QRS_NEXT_CUT()
PTP {E1 28976.919,E2 28976.919}
PTP {X 0,Y 607.89,A -85,B 0,C 180,E1 28976.919,E2 28976.919,E3 0,E4 0,E5 0,E6 0}
QRS_SPEED_INIT()
LIN {X 0,Y 607.89,Z 1319.5,A -85,B 0,C 180,E1 28976.919,E2 28976.919,E3 0,E4 0,E5 0,E6 0} C_VEL
LIN {X 0,Y 607.89,Z 669.091,A -85,B 0,C 180,E1 28976.919,E2 28976.919} C_VEL
LIN {X 0,Y 607.89,Z 661.015,A -85,B 0,C 180,E1 28976.919,E2 28976.919} C_VEL
LIN {X 0,Y 607.896,Z 659.015,A -85,B 0,C 180,E1 28976.73,E2 28976.73} C_VEL
LIN {X 0,Y 607.914,Z 659.013,A -85,B 0,C 180,E1 28973.578,E2 28973.578} C_VEL
LIN {X 0,Y 607.913,Z 659.015,A -85,B 0,C 180,E1 28970.342,E2 28970.342} C_VEL
LIN {X 0,Y 607.906,Z 659.015,A -85,B 0,C 180,E1 28967.171,E2 28967.171} C_VEL
LIN {X 0,Y 607.906,Z 659.013,A -85,B 0,C 180,E1 28963.959,E2 28963.959} C_VEL
LIN {X 0,Y 607.896,Z 659.013,A -85,B 0,C 180,E1 28960.751,E2 28960.751} C_VEL
LIN {X 0,Y 607.9,Z 659.012,A -85,B 0,C 180,E1 28957.67,E2 28957.67} C_VEL
LIN {X 0,Y 607.904,Z 659.011,A -85,B 0,C 180,E1 28954.473,E2 28954.473} C_VEL
LIN {X 0,Y 607.904,Z 659.009,A -85,B 0,C 180,E1 28951.241,E2 28951.241} C_VEL
LIN {X 0,Y 607.906,Z 659.01,A -85,B 0,C 180,E1 28948.021,E2 28948.021} C_VEL
LIN {X 0,Y 607.908,Z 659.009,A -85,B 0,C 180,E1 28944.828,E2 28944.828} C_VEL
LIN {X 0,Y 607.911,Z 659.01,A -85,B 0,C 180,E1 28941.526,E2 28941.526} C_VEL
LIN {X 0,Y 607.907,Z 659.011,A -85,B 0,C 180,E1 28938.306,E2 28938.306} C_VEL
LIN {X 0,Y 607.917,Z 659.013,A -85,B 0,C 180,E1 28935.009,E2 28935.009} C_VEL
LIN {X 0,Y 607.911,Z 659.016,A -85,B 0,C 180,E1 28931.768,E2 28931.768} C_VEL
LIN {X 0,Y 607.904,Z 659.015,A -85,B 0,C 180,E1 28928.562,E2 28928.562} C_VEL
LIN {X 0,Y 607.904,Z 659.014,A -85,B 0,C 180,E1 28925.376,E2 28925.376} C_VEL
LIN {X 0,Y 607.916,Z 659.13,A -85,B 0,C 180,E1 28924.285,E2 28924.285} C_VEL
LIN {X 0,Y 607.915,Z 707.559,A -85,B 0,C 180,E1 28921.204,E2 28921.204} C_VEL
LIN {X 0,Y 607.914,Z 757.754,A -85,B 0,C 180,E1 28918.113,E2 28918.113} C_VEL
LIN {X 0,Y 607.895,Z 765.812,A -85,B 0,C 180,E1 28917.641,E2 28917.641} C_VEL
LIN {X 0,Y 607.908,Z 1003.67,A -85,B 0,C 180,E1 28914.573,E2 28914.573} C_VEL
LIN {X 0,Y 607.919,Z 1031.222,A -85,B 0,C 180,E1 28914.175,E2 28914.175} C_VEL
LIN {X 0,Y 607.917,Z 1051.471,A -85,B 0,C 180,E1 28913.711,E2 28913.711} C_VEL
LIN {X 0,Y 607.906,Z 1071.416,A -85,B 0,C 180,E1 28913.07,E2 28913.07} C_VEL
LIN {X 0,Y 607.906,Z 1090.488,A -85,B 0,C 180,E1 28912.278,E2 28912.278} C_VEL
LIN {X 0,Y 607.918,Z 1109.332,A -85,B 0,C 180,E1 28911.314,E2 28911.314} C_VEL
LIN {X 0,Y 607.917,Z 1127.307,A -85,B 0,C 180,E1 28910.205,E2 28910.205} C_VEL
LIN {X 0,Y 607.912,Z 1144.273,A -85,B 0,C 180,E1 28908.963,E2 28908.963} C_VEL
LIN {X 0,Y 607.917,Z 1160.452,A -85,B 0,C 180,E1 28907.566,E2 28907.566} C_VEL
LIN {X 0,Y 607.913,Z 1175.45,A -85,B 0,C 180,E1 28906.04,E2 28906.04} C_VEL
LIN {X 0,Y 607.913,Z 1189.435,A -85,B 0,C 180,E1 28904.36,E2 28904.36} C_VEL
LIN {X 0,Y 607.909,Z 1201.499,A -85,B 0,C 180,E1 28902.635,E2 28902.635} C_VEL
LIN {X 0,Y 607.917,Z 1211.62,A -85,B 0,C 180,E1 28900.902,E2 28900.902} C_VEL
LIN {X 0,Y 607.904,Z 1220.371,A -85,B 0,C 180,E1 28899.084,E2 28899.084} C_VEL
LIN {X 0,Y 607.901,Z 1227.349,A -85,B 0,C 180,E1 28897.275,E2 28897.275} C_VEL
LIN {X 0,Y 607.911,Z 1232.888,A -85,B 0,C 180,E1 28895.379,E2 28895.379} C_VEL
LIN {X 0,Y 607.905,Z 1236.665,A -85,B 0,C 180,E1 28893.489,E2 28893.489} C_VEL
LIN {X 0,Y 607.904,Z 1238.841,A -85,B 0,C 180,E1 28891.602,E2 28891.602} C_VEL
LIN {X 0,Y 607.904,Z 1239.45,A -85,B 0,C 180,E1 28889.717,E2 28889.717} C_VEL
LIN {X 0,Y 607.919,Z 1238.497,A -85,B 0,C 180,E1 28887.832,E2 28887.832} C_VEL
LIN {X 0,Y 607.916,Z 1235.709,A -85,B 0,C 180,E1 28885.85,E2 28885.85} C_VEL
LIN {X 0,Y 607.91,Z 1231.354,A -85,B 0,C 180,E1 28883.957,E2 28883.957} C_VEL
LIN {X 0,Y 607.904,Z 1225.285,A -85,B 0,C 180,E1 28882.058,E2 28882.058} C_VEL
LIN {X 0,Y 607.911,Z 1217.814,A -85,B 0,C 180,E1 28880.246,E2 28880.246} C_VEL
LIN {X 0,Y 607.907,Z 1208.471,A -85,B 0,C 180,E1 28878.424,E2 28878.424} C_VEL
LIN {X 0,Y 607.906,Z 1197.61,A -85,B 0,C 180,E1 28876.687,E2 28876.687} C_VEL
LIN {X 0,Y 607.914,Z 1185.34,A -85,B 0,C 180,E1 28875.035,E2 28875.035} C_VEL
LIN {X 0,Y 607.916,Z 1171.664,A -85,B 0,C 180,E1 28873.468,E2 28873.468} C_VEL
LIN {X 0,Y 607.912,Z 1156.498,A -85,B 0,C 180,E1 28871.988,E2 28871.988} C_VEL
LIN {X 0,Y 607.918,Z 1139.693,A -85,B 0,C 180,E1 28870.595,E2 28870.595} C_VEL
LIN {X 0,Y 607.917,Z 1122.559,A -85,B 0,C 180,E1 28869.392,E2 28869.392} C_VEL
LIN {X 0,Y 607.918,Z 1104.436,A -85,B 0,C 180,E1 28868.322,E2 28868.322} C_VEL
LIN {X 0,Y 607.916,Z 1085.73,A -85,B 0,C 180,E1 28867.415,E2 28867.415} C_VEL
LIN {X 0,Y 607.911,Z 1066.623,A -85,B 0,C 180,E1 28866.673,E2 28866.673} C_VEL
LIN {X 0,Y 607.913,Z 1045.815,A -85,B 0,C 180,E1 28866.055,E2 28866.055} C_VEL
LIN {X 0,Y 607.911,Z 1026.135,A -85,B 0,C 180,E1 28865.644,E2 28865.644} C_VEL
LIN {X 0,Y 607.897,Z 777.541,A -85,B 0,C 180,E1 28862.423,E2 28862.423} C_VEL
LIN {X 0,Y 607.904,Z 767.538,A -85,B 0,C 180,E1 28862.286,E2 28862.286} C_VEL
LIN {X 0,Y 607.9,Z 733.072,A -85,B 0,C 180,E1 28859.287,E2 28859.287} C_VEL
LIN {X 0,Y 607.898,Z 699.537,A -85,B 0,C 180,E1 28856.278,E2 28856.278} C_VEL
LIN {X 0,Y 607.908,Z 666.674,A -85,B 0,C 180,E1 28853.224,E2 28853.224} C_VEL
LIN {X 0,Y 607.903,Z 659.012,A -85,B 0,C 180,E1 28852.48,E2 28852.48} C_VEL
LIN {X 0,Y 607.907,Z 659.006,A -85,B 0,C 180,E1 28849.234,E2 28849.234} C_VEL
LIN {X 0,Y 607.918,Z 659.015,A -85,B 0,C 180,E1 28845.915,E2 28845.915} C_VEL
LIN {X 0,Y 607.909,Z 659.005,A -85,B 0,C 180,E1 28842.66,E2 28842.66} C_VEL
LIN {X 0,Y 607.912,Z 659.007,A -85,B 0,C 180,E1 28839.289,E2 28839.289} C_VEL
LIN {X 0,Y 607.917,Z 659.013,A -85,B 0,C 180,E1 28835.957,E2 28835.957} C_VEL
LIN {X 0,Y 607.902,Z 659.007,A -85,B 0,C 180,E1 28832.649,E2 28832.649} C_VEL
LIN {X 0,Y 607.893,Z 659.115,A -85,B 0,C 180,E1 28831.289,E2 28831.289} C_VEL
LIN {X 0,Y 607.901,Z 697.133,A -85,B 0,C 180,E1 28828.319,E2 28828.319} C_VEL
LIN {X 0,Y 607.908,Z 738.09,A -85,B 0,C 180,E1 28825.214,E2 28825.214} C_VEL
LIN {X 0,Y 607.909,Z 781.964,A -85,B 0,C 180,E1 28821.977,E2 28821.977} C_VEL
LIN {X 0,Y 607.917,Z 826.671,A -85,B 0,C 180,E1 28818.757,E2 28818.757} C_VEL
LIN {X 0,Y 607.898,Z 844.902,A -85,B 0,C 180,E1 28817.467,E2 28817.467} C_VEL
LIN {X 0,Y 607.901,Z 1015.001,A -85,B 0,C 180,E1 28815.38,E2 28815.38} C_VEL
LIN {X 0,Y 607.917,Z 1032.362,A -85,B 0,C 180,E1 28814.989,E2 28814.989} C_VEL
LIN {X 0,Y 607.915,Z 1049.263,A -85,B 0,C 180,E1 28814.429,E2 28814.429} C_VEL
LIN {X 0,Y 607.905,Z 1065.628,A -85,B 0,C 180,E1 28813.701,E2 28813.701} C_VEL
LIN {X 0,Y 607.919,Z 1080.913,A -85,B 0,C 180,E1 28812.829,E2 28812.829} C_VEL
LIN {X 0,Y 607.917,Z 1095.13,A -85,B 0,C 180,E1 28811.816,E2 28811.816} C_VEL
LIN {X 0,Y 607.915,Z 1108.876,A -85,B 0,C 180,E1 28810.615,E2 28810.615} C_VEL
LIN {X 0,Y 607.915,Z 1120.53,A -85,B 0,C 180,E1 28809.371,E2 28809.371} C_VEL
LIN {X 0,Y 607.918,Z 1130.726,A -85,B 0,C 180,E1 28808.037,E2 28808.037} C_VEL
LIN {X 0,Y 607.913,Z 1139.724,A -85,B 0,C 180,E1 28806.574,E2 28806.574} C_VEL
LIN {X 0,Y 607.916,Z 1147.292,A -85,B 0,C 180,E1 28805.001,E2 28805.001} C_VEL
LIN {X 0,Y 607.915,Z 1153.026,A -85,B 0,C 180,E1 28803.395,E2 28803.395} C_VEL
LIN {X 0,Y 607.913,Z 1156.875,A -85,B 0,C 180,E1 28801.791,E2 28801.791} C_VEL
LIN {X 0,Y 607.913,Z 1158.976,A -85,B 0,C 180,E1 28800.189,E2 28800.189} C_VEL
LIN {X 0,Y 607.913,Z 1159.398,A -85,B 0,C 180,E1 28798.492,E2 28798.492} C_VEL
LIN {X 0,Y 607.91,Z 1157.985,A -85,B 0,C 180,E1 28796.794,E2 28796.794} C_VEL
LIN {X 0,Y 607.918,Z 1154.852,A -85,B 0,C 180,E1 28795.189,E2 28795.189} C_VEL
LIN {X 0,Y 607.912,Z 1149.903,A -85,B 0,C 180,E1 28793.579,E2 28793.579} C_VEL
LIN {X 0,Y 607.912,Z 1142.996,A -85,B 0,C 180,E1 28791.964,E2 28791.964} C_VEL
LIN {X 0,Y 607.914,Z 1134.47,A -85,B 0,C 180,E1 28790.438,E2 28790.438} C_VEL
LIN {X 0,Y 607.917,Z 1124.947,A -85,B 0,C 180,E1 28789.084,E2 28789.084} C_VEL
LIN {X 0,Y 607.915,Z 1113.389,A -85,B 0,C 180,E1 28787.751,E2 28787.751} C_VEL
LIN {X 0,Y 607.917,Z 1100.614,A -85,B 0,C 180,E1 28786.542,E2 28786.542} C_VEL
LIN {X 0,Y 607.918,Z 1086.802,A -85,B 0,C 180,E1 28785.474,E2 28785.474} C_VEL
LIN {X 0,Y 607.914,Z 1071.813,A -85,B 0,C 180,E1 28784.54,E2 28784.54} C_VEL
LIN {X 0,Y 607.912,Z 1056.138,A -85,B 0,C 180,E1 28783.764,E2 28783.764} C_VEL
LIN {X 0,Y 607.912,Z 1039.216,A -85,B 0,C 180,E1 28783.124,E2 28783.124} C_VEL
LIN {X 0,Y 607.912,Z 1022.717,A -85,B 0,C 180,E1 28782.681,E2 28782.681} C_VEL
LIN {X 0,Y 607.912,Z 1004.843,A -85,B 0,C 180,E1 28782.384,E2 28782.384} C_VEL
LIN {X 0,Y 607.899,Z 844.692,A -85,B 0,C 180,E1 28780.432,E2 28780.432} C_VEL
LIN {X 0,Y 607.912,Z 800.299,A -85,B 0,C 180,E1 28777.262,E2 28777.262} C_VEL
LIN {X 0,Y 607.894,Z 758.501,A -85,B 0,C 180,E1 28774.212,E2 28774.212} C_VEL
LIN {X 0,Y 607.901,Z 718.072,A -85,B 0,C 180,E1 28771.189,E2 28771.189} C_VEL
LIN {X 0,Y 607.915,Z 677.489,A -85,B 0,C 180,E1 28768.069,E2 28768.069} C_VEL
LIN {X 0,Y 607.898,Z 659.016,A -85,B 0,C 180,E1 28766.591,E2 28766.591} C_VEL
LIN {X 0,Y 607.894,Z 659.014,A -85,B 0,C 180,E1 28763.458,E2 28763.458} C_VEL
LIN {X 0,Y 607.916,Z 659.015,A -85,B 0,C 180,E1 28760.33,E2 28760.33} C_VEL
LIN {X 0,Y 607.906,Z 659.143,A -85,B 0,C 180,E1 28759.424,E2 28759.424} C_VEL
LIN {X 0,Y 607.915,Z 712.703,A -85,B 0,C 180,E1 28757.135,E2 28757.135} C_VEL
LIN {X 0,Y 607.918,Z 729.762,A -85,B 0,C 180,E1 28756.308,E2 28756.308} C_VEL
LIN {X 0,Y 607.904,Z 743.335,A -85,B 0,C 180,E1 28755.466,E2 28755.466} C_VEL
LIN {X 0,Y 607.911,Z 752.379,A -85,B 0,C 180,E1 28754.722,E2 28754.722} C_VEL
LIN {X 0,Y 607.912,Z 757.786,A -85,B 0,C 180,E1 28754.085,E2 28754.085} C_VEL
LIN {X 0,Y 607.908,Z 759.997,A -85,B 0,C 180,E1 28753.64,E2 28753.64} C_VEL
LIN {X 0,Y 607.915,Z 760.434,A -85,B 0,C 180,E1 28753.23,E2 28753.23} C_VEL
LIN {X 0,Y 607.904,Z 759.309,A -85,B 0,C 180,E1 28752.917,E2 28752.917} C_VEL
LIN {X 0,Y 607.894,Z 756.773,A -85,B 0,C 180,E1 28752.661,E2 28752.661} C_VEL
LIN {X 0,Y 607.9,Z 751.993,A -85,B 0,C 180,E1 28752.437,E2 28752.437} C_VEL
LIN {X 0,Y 607.912,Z 744.111,A -85,B 0,C 180,E1 28752.283,E2 28752.283} C_VEL
LIN {X 0,Y 607.916,Z 737.218,A -85,B 0,C 180,E1 28752.249,E2 28752.249} C_VEL
LIN {X 0,Y 607.916,Z 659.014,A -85,B 0,C 180,E1 28752.23,E2 28752.23} C_VEL
LIN {X 0,Y 607.906,Z 659.014,A -85,B 0,C 180,E1 28748.925,E2 28748.925} C_VEL
LIN {X 0,Y 607.903,Z 659.112,A -85,B 0,C 180,E1 28748.115,E2 28748.115} C_VEL
LIN {X 0,Y 607.899,Z 707.786,A -85,B 0,C 180,E1 28745.262,E2 28745.262} C_VEL
LIN {X 0,Y 607.911,Z 759.02,A -85,B 0,C 180,E1 28742.372,E2 28742.372} C_VEL
LIN {X 0,Y 607.915,Z 990.402,A -85,B 0,C 180,E1 28739.254,E2 28739.254} C_VEL
LIN {X 0,Y 607.906,Z 1065.532,A -85,B 0,C 180,E1 28738.234,E2 28738.234} C_VEL
LIN {X 0,Y 607.913,Z 1086.021,A -85,B 0,C 180,E1 28737.786,E2 28737.786} C_VEL
LIN {X 0,Y 607.909,Z 1106.622,A -85,B 0,C 180,E1 28737.18,E2 28737.18} C_VEL
LIN {X 0,Y 607.904,Z 1126.576,A -85,B 0,C 180,E1 28736.418,E2 28736.418} C_VEL
LIN {X 0,Y 607.918,Z 1147.741,A -85,B 0,C 180,E1 28735.422,E2 28735.422} C_VEL
LIN {X 0,Y 607.916,Z 1167.109,A -85,B 0,C 180,E1 28734.332,E2 28734.332} C_VEL
LIN {X 0,Y 607.914,Z 1185.555,A -85,B 0,C 180,E1 28733.096,E2 28733.096} C_VEL
LIN {X 0,Y 607.913,Z 1203.767,A -85,B 0,C 180,E1 28731.678,E2 28731.678} C_VEL
LIN {X 0,Y 607.915,Z 1220.646,A -85,B 0,C 180,E1 28730.156,E2 28730.156} C_VEL
LIN {X 0,Y 607.918,Z 1236.463,A -85,B 0,C 180,E1 28728.508,E2 28728.508} C_VEL
LIN {X 0,Y 607.912,Z 1251.11,A -85,B 0,C 180,E1 28726.728,E2 28726.728} C_VEL
LIN {X 0,Y 607.911,Z 1263.539,A -85,B 0,C 180,E1 28724.965,E2 28724.965} C_VEL
LIN {X 0,Y 607.918,Z 1275.248,A -85,B 0,C 180,E1 28723.022,E2 28723.022} C_VEL
LIN {X 0,Y 607.914,Z 1284.984,A -85,B 0,C 180,E1 28721.095,E2 28721.095} C_VEL
LIN {X 0,Y 607.909,Z 1292.817,A -85,B 0,C 180,E1 28719.181,E2 28719.181} C_VEL
LIN {X 0,Y 607.905,Z 1299.381,A -85,B 0,C 180,E1 28717.181,E2 28717.181} C_VEL
LIN {X 0,Y 607.911,Z 1304.014,A -85,B 0,C 180,E1 28715.285,E2 28715.285} C_VEL
LIN {X 0,Y 607.916,Z 1307.446,A -85,B 0,C 180,E1 28713.206,E2 28713.206} C_VEL
LIN {X 0,Y 607.91,Z 1309.209,A -85,B 0,C 180,E1 28711.226,E2 28711.226} C_VEL
LIN {X 0,Y 607.897,Z 1309.329,A -85,B 0,C 180,E1 28709.246,E2 28709.246} C_VEL
LIN {X 0,Y 607.897,Z 1307.896,A -85,B 0,C 180,E1 28707.172,E2 28707.172} C_VEL
LIN {X 0,Y 607.902,Z 1304.988,A -85,B 0,C 180,E1 28705.189,E2 28705.189} C_VEL
LIN {X 0,Y 607.912,Z 1300.399,A -85,B 0,C 180,E1 28703.199,E2 28703.199} C_VEL
LIN {X 0,Y 607.909,Z 1294.24,A -85,B 0,C 180,E1 28701.202,E2 28701.202} C_VEL
LIN {X 0,Y 607.909,Z 1286.659,A -85,B 0,C 180,E1 28699.289,E2 28699.289} C_VEL
LIN {X 0,Y 607.9,Z 1277.329,A -85,B 0,C 180,E1 28697.365,E2 28697.365} C_VEL
LIN {X 0,Y 607.901,Z 1266.748,A -85,B 0,C 180,E1 28695.523,E2 28695.523} C_VEL
LIN {X 0,Y 607.909,Z 1254.038,A -85,B 0,C 180,E1 28693.666,E2 28693.666} C_VEL
LIN {X 0,Y 607.912,Z 1239.872,A -85,B 0,C 180,E1 28691.89,E2 28691.89} C_VEL
LIN {X 0,Y 607.91,Z 1224.091,A -85,B 0,C 180,E1 28690.185,E2 28690.185} C_VEL
LIN {X 0,Y 607.915,Z 1207.506,A -85,B 0,C 180,E1 28688.636,E2 28688.636} C_VEL
LIN {X 0,Y 607.913,Z 1189.143,A -85,B 0,C 180,E1 28687.161,E2 28687.161} C_VEL
LIN {X 0,Y 607.916,Z 1170.68,A -85,B 0,C 180,E1 28685.898,E2 28685.898} C_VEL
LIN {X 0,Y 607.917,Z 1150.562,A -85,B 0,C 180,E1 28684.726,E2 28684.726} C_VEL
LIN {X 0,Y 607.9,Z 1130.391,A -85,B 0,C 180,E1 28683.741,E2 28683.741} C_VEL
LIN {X 0,Y 607.914,Z 1110.253,A -85,B 0,C 180,E1 28682.951,E2 28682.951} C_VEL
LIN {X 0,Y 607.915,Z 1087.821,A -85,B 0,C 180,E1 28682.261,E2 28682.261} C_VEL
LIN {X 0,Y 607.907,Z 1067.099,A -85,B 0,C 180,E1 28681.793,E2 28681.793} C_VEL
LIN {X 0,Y 607.913,Z 1025.867,A -85,B 0,C 180,E1 28681.215,E2 28681.215} C_VEL
LIN {X 0,Y 607.892,Z 804.134,A -85,B 0,C 180,E1 28678.243,E2 28678.243} C_VEL
LIN {X 0,Y 607.913,Z 758.441,A -85,B 0,C 180,E1 28677.604,E2 28677.604} C_VEL
LIN {X 0,Y 607.912,Z 702.746,A -85,B 0,C 180,E1 28674.448,E2 28674.448} C_VEL
LIN {X 0,Y 607.903,Z 659.014,A -85,B 0,C 180,E1 28671.875,E2 28671.875} C_VEL
LIN {X 0,Y 607.901,Z 659.015,A -85,B 0,C 180,E1 28668.734,E2 28668.734} C_VEL
LIN {X 0,Y 607.916,Z 659.014,A -85,B 0,C 180,E1 28667.752,E2 28667.752} C_VEL
LIN {X 0,Y 607.914,Z 742.107,A -85,B 0,C 180,E1 28667.734,E2 28667.734} C_VEL
LIN {X 0,Y 607.902,Z 750.866,A -85,B 0,C 180,E1 28667.597,E2 28667.597} C_VEL
LIN {X 0,Y 607.894,Z 755.763,A -85,B 0,C 180,E1 28667.403,E2 28667.403} C_VEL
LIN {X 0,Y 607.899,Z 758.521,A -85,B 0,C 180,E1 28667.186,E2 28667.186} C_VEL
LIN {X 0,Y 607.915,Z 760.123,A -85,B 0,C 180,E1 28666.908,E2 28666.908} C_VEL
LIN {X 0,Y 607.917,Z 760.432,A -85,B 0,C 180,E1 28666.569,E2 28666.569} C_VEL
LIN {X 0,Y 607.906,Z 758.831,A -85,B 0,C 180,E1 28666.087,E2 28666.087} C_VEL
LIN {X 0,Y 607.916,Z 754.212,A -85,B 0,C 180,E1 28665.466,E2 28665.466} C_VEL
LIN {X 0,Y 607.914,Z 746.157,A -85,B 0,C 180,E1 28664.744,E2 28664.744} C_VEL
LIN {X 0,Y 607.913,Z 732.359,A -85,B 0,C 180,E1 28663.823,E2 28663.823} C_VEL
LIN {X 0,Y 607.914,Z 692.649,A -85,B 0,C 180,E1 28661.264,E2 28661.264} C_VEL
LIN {X 0,Y 607.896,Z 659.012,A -85,B 0,C 180,E1 28658.971,E2 28658.971} C_VEL
LIN {X 0,Y 607.9,Z 659.011,A -85,B 0,C 180,E1 28655.82,E2 28655.82} C_VEL
LIN {X 0,Y 607.906,Z 659.01,A -85,B 0,C 180,E1 28652.637,E2 28652.637} C_VEL
LIN {X 0,Y 607.905,Z 659.011,A -85,B 0,C 180,E1 28649.458,E2 28649.458} C_VEL
LIN {X 0,Y 607.914,Z 659.01,A -85,B 0,C 180,E1 28646.259,E2 28646.259} C_VEL
LIN {X 0,Y 607.91,Z 659.012,A -85,B 0,C 180,E1 28643.045,E2 28643.045} C_VEL
LIN {X 0,Y 607.918,Z 659.013,A -85,B 0,C 180,E1 28639.804,E2 28639.804} C_VEL
LIN {X 0,Y 607.916,Z 659.015,A -85,B 0,C 180,E1 28636.531,E2 28636.531} C_VEL
LIN {X 0,Y 607.905,Z 659.014,A -85,B 0,C 180,E1 28633.313,E2 28633.313} C_VEL
LIN {X 0,Y 607.911,Z 659.012,A -85,B 0,C 180,E1 28630.136,E2 28630.136} C_VEL
LIN {X 0,Y 607.91,Z 659.01,A -85,B 0,C 180,E1 28626.896,E2 28626.896} C_VEL
LIN {X 0,Y 607.909,Z 659.01,A -85,B 0,C 180,E1 28623.678,E2 28623.678} C_VEL
LIN {X 0,Y 607.908,Z 659.009,A -85,B 0,C 180,E1 28620.377,E2 28620.377} C_VEL
LIN {X 0,Y 607.909,Z 659.01,A -85,B 0,C 180,E1 28617.172,E2 28617.172} C_VEL
LIN {X 0,Y 607.896,Z 659.015,A -85,B 0,C 180,E1 28616.73,E2 28616.73} C_VEL
LIN {X 0,Y 606.924,Z 659.142,A -85,B 0,C 180,E1 28616.004,E2 28616.004} C_VEL
LIN {X 0,Y 600.428,Z 659.947,A -85,B 0,C 180,E1 28613.915,E2 28613.915} C_VEL
LIN {X 0,Y 599.972,Z 660.004,A -85,B 0,C 180,E1 28613.437,E2 28613.437} C_VEL
LIN {X 0,Y 599.974,Z 660.002,A -85,B 0,C 180,E1 28610.213,E2 28610.213} C_VEL
LIN {X 0,Y 599.955,Z 660.003,A -85,B 0,C 180,E1 28606.998,E2 28606.998} C_VEL
LIN {X 0,Y 599.964,Z 660.001,A -85,B 0,C 180,E1 28603.84,E2 28603.84} C_VEL
LIN {X 0,Y 599.955,Z 660.001,A -85,B 0,C 180,E1 28600.631,E2 28600.631} C_VEL
LIN {X 0,Y 599.957,Z 660.001,A -85,B 0,C 180,E1 28597.564,E2 28597.564} C_VEL
LIN {X 0,Y 599.959,Z 660,A -85,B 0,C 180,E1 28594.368,E2 28594.368} C_VEL
LIN {X 0,Y 599.963,Z 659.996,A -85,B 0,C 180,E1 28591.208,E2 28591.208} C_VEL
LIN {X 0,Y 599.966,Z 659.999,A -85,B 0,C 180,E1 28587.997,E2 28587.997} C_VEL
LIN {X 0,Y 599.963,Z 659.997,A -85,B 0,C 180,E1 28584.745,E2 28584.745} C_VEL
LIN {X 0,Y 599.973,Z 659.999,A -85,B 0,C 180,E1 28581.559,E2 28581.559} C_VEL
LIN {X 0,Y 599.969,Z 659.999,A -85,B 0,C 180,E1 28578.296,E2 28578.296} C_VEL
LIN {X 0,Y 599.978,Z 660.002,A -85,B 0,C 180,E1 28575.041,E2 28575.041} C_VEL
LIN {X 0,Y 599.972,Z 660.005,A -85,B 0,C 180,E1 28571.805,E2 28571.805} C_VEL
LIN {X 0,Y 599.965,Z 660.004,A -85,B 0,C 180,E1 28568.555,E2 28568.555} C_VEL
LIN {X 0,Y 599.967,Z 660.004,A -85,B 0,C 180,E1 28565.419,E2 28565.419} C_VEL
LIN {X 0,Y 599.965,Z 660.024,A -85,B 0,C 180,E1 28564.746,E2 28564.746} C_VEL
LIN {X 0,Y 600.946,Z 663.544,A -85,B 0,C 180,E1 28564.45,E2 28564.45} C_VEL
LIN {X 0,Y 600.77,Z 711.4,A -85,B 0,C 180,E1 28561.374,E2 28561.374} C_VEL
LIN {X 0,Y 600.618,Z 761.087,A -85,B 0,C 180,E1 28558.281,E2 28558.281} C_VEL
LIN {X 0,Y 600.684,Z 766.073,A -85,B 0,C 180,E1 28557.999,E2 28557.999} C_VEL
LIN {X 0,Y 600.669,Z 957.534,A -85,B 0,C 180,E1 28555.487,E2 28555.487} C_VEL
LIN {X 0,Y 600.612,Z 1028.42,A -85,B 0,C 180,E1 28554.544,E2 28554.544} C_VEL
LIN {X 0,Y 600.567,Z 1049.119,A -85,B 0,C 180,E1 28554.083,E2 28554.083} C_VEL
LIN {X 0,Y 600.495,Z 1069.241,A -85,B 0,C 180,E1 28553.449,E2 28553.449} C_VEL
LIN {X 0,Y 600.42,Z 1088.269,A -85,B 0,C 180,E1 28552.675,E2 28552.675} C_VEL
LIN {X 0,Y 600.347,Z 1106.872,A -85,B 0,C 180,E1 28551.739,E2 28551.739} C_VEL
LIN {X 0,Y 600.277,Z 1125.207,A -85,B 0,C 180,E1 28550.622,E2 28550.622} C_VEL
LIN {X 0,Y 600.196,Z 1143.319,A -85,B 0,C 180,E1 28549.295,E2 28549.295} C_VEL
LIN {X 0,Y 600.123,Z 1159.921,A -85,B 0,C 180,E1 28547.852,E2 28547.852} C_VEL
LIN {X 0,Y 600.063,Z 1174.973,A -85,B 0,C 180,E1 28546.308,E2 28546.308} C_VEL
LIN {X 0,Y 600.007,Z 1188.517,A -85,B 0,C 180,E1 28544.672,E2 28544.672} C_VEL
LIN {X 0,Y 599.977,Z 1200.227,A -85,B 0,C 180,E1 28543.001,E2 28543.001} C_VEL
LIN {X 0,Y 599.947,Z 1211.108,A -85,B 0,C 180,E1 28541.146,E2 28541.146} C_VEL
LIN {X 0,Y 599.925,Z 1219.968,A -85,B 0,C 180,E1 28539.303,E2 28539.303} C_VEL
LIN {X 0,Y 599.919,Z 1227.049,A -85,B 0,C 180,E1 28537.469,E2 28537.469} C_VEL
LIN {X 0,Y 599.917,Z 1232.637,A -85,B 0,C 180,E1 28535.547,E2 28535.547} C_VEL
LIN {X 0,Y 599.908,Z 1236.508,A -85,B 0,C 180,E1 28533.631,E2 28533.631} C_VEL
LIN {X 0,Y 599.905,Z 1238.842,A -85,B 0,C 180,E1 28531.623,E2 28531.623} C_VEL
LIN {X 0,Y 599.904,Z 1239.45,A -85,B 0,C 180,E1 28529.713,E2 28529.713} C_VEL
LIN {X 0,Y 599.917,Z 1238.497,A -85,B 0,C 180,E1 28527.803,E2 28527.803} C_VEL
LIN {X 0,Y 599.917,Z 1235.708,A -85,B 0,C 180,E1 28525.794,E2 28525.794} C_VEL
LIN {X 0,Y 599.912,Z 1231.353,A -85,B 0,C 180,E1 28523.876,E2 28523.876} C_VEL
LIN {X 0,Y 599.91,Z 1225.076,A -85,B 0,C 180,E1 28521.895,E2 28521.895} C_VEL
LIN {X 0,Y 599.924,Z 1217.351,A -85,B 0,C 180,E1 28520.018,E2 28520.018} C_VEL
LIN {X 0,Y 599.948,Z 1208.468,A -85,B 0,C 180,E1 28518.268,E2 28518.268} C_VEL
LIN {X 0,Y 599.971,Z 1197.609,A -85,B 0,C 180,E1 28516.508,E2 28516.508} C_VEL
LIN {X 0,Y 600.02,Z 1185.338,A -85,B 0,C 180,E1 28514.833,E2 28514.833} C_VEL
LIN {X 0,Y 600.065,Z 1171.661,A -85,B 0,C 180,E1 28513.246,E2 28513.246} C_VEL
LIN {X 0,Y 600.132,Z 1155.941,A -85,B 0,C 180,E1 28511.696,E2 28511.696} C_VEL
LIN {X 0,Y 600.206,Z 1139.687,A -85,B 0,C 180,E1 28510.336,E2 28510.336} C_VEL
LIN {X 0,Y 600.289,Z 1122.551,A -85,B 0,C 180,E1 28509.118,E2 28509.118} C_VEL
LIN {X 0,Y 600.37,Z 1104.598,A -85,B 0,C 180,E1 28508.044,E2 28508.044} C_VEL
LIN {X 0,Y 600.434,Z 1085.722,A -85,B 0,C 180,E1 28507.118,E2 28507.118} C_VEL
LIN {X 0,Y 600.502,Z 1066.613,A -85,B 0,C 180,E1 28506.368,E2 28506.368} C_VEL
LIN {X 0,Y 600.569,Z 1045.951,A -85,B 0,C 180,E1 28505.748,E2 28505.748} C_VEL
LIN {X 0,Y 600.616,Z 1025.33,A -85,B 0,C 180,E1 28505.316,E2 28505.316} C_VEL
LIN {X 0,Y 600.8,Z 778.085,A -85,B 0,C 180,E1 28502.077,E2 28502.077} C_VEL
LIN {X 0,Y 600.581,Z 768.202,A -85,B 0,C 180,E1 28501.934,E2 28501.934} C_VEL
LIN {X 0,Y 600.471,Z 765.978,A -85,B 0,C 180,E1 28501.777,E2 28501.777} C_VEL
LIN {X 0,Y 600.6,Z 729.358,A -85,B 0,C 180,E1 28498.54,E2 28498.54} C_VEL
LIN {X 0,Y 600.733,Z 694.016,A -85,B 0,C 180,E1 28495.307,E2 28495.307} C_VEL
LIN {X 0,Y 600.833,Z 662.738,A -85,B 0,C 180,E1 28492.338,E2 28492.338} C_VEL
LIN {X 0,Y 599.974,Z 660.005,A -85,B 0,C 180,E1 28491.992,E2 28491.992} C_VEL
LIN {X 0,Y 599.959,Z 659.997,A -85,B 0,C 180,E1 28488.73,E2 28488.73} C_VEL
LIN {X 0,Y 599.964,Z 660,A -85,B 0,C 180,E1 28485.577,E2 28485.577} C_VEL
LIN {X 0,Y 599.974,Z 659.996,A -85,B 0,C 180,E1 28482.416,E2 28482.416} C_VEL
LIN {X 0,Y 599.967,Z 659.996,A -85,B 0,C 180,E1 28479.169,E2 28479.169} C_VEL
LIN {X 0,Y 599.978,Z 660.004,A -85,B 0,C 180,E1 28475.912,E2 28475.912} C_VEL
LIN {X 0,Y 599.966,Z 659.997,A -85,B 0,C 180,E1 28472.681,E2 28472.681} C_VEL
LIN {X 0,Y 599.975,Z 660.054,A -85,B 0,C 180,E1 28471.693,E2 28471.693} C_VEL
LIN {X 0,Y 600.692,Z 663.62,A -85,B 0,C 180,E1 28471.362,E2 28471.362} C_VEL
LIN {X 0,Y 600.559,Z 701.404,A -85,B 0,C 180,E1 28468.381,E2 28468.381} C_VEL
LIN {X 0,Y 600.437,Z 741.833,A -85,B 0,C 180,E1 28465.282,E2 28465.282} C_VEL
LIN {X 0,Y 600.324,Z 784.307,A -85,B 0,C 180,E1 28462.112,E2 28462.112} C_VEL
LIN {X 0,Y 600.227,Z 828.974,A -85,B 0,C 180,E1 28458.855,E2 28458.855} C_VEL
LIN {X 0,Y 600.24,Z 845.305,A -85,B 0,C 180,E1 28457.707,E2 28457.707} C_VEL
LIN {X 0,Y 600.22,Z 1015.448,A -85,B 0,C 180,E1 28455.588,E2 28455.588} C_VEL
LIN {X 0,Y 600.208,Z 1033.412,A -85,B 0,C 180,E1 28455.171,E2 28455.171} C_VEL
LIN {X 0,Y 600.17,Z 1049.631,A -85,B 0,C 180,E1 28454.619,E2 28454.619} C_VEL
LIN {X 0,Y 600.117,Z 1064.926,A -85,B 0,C 180,E1 28453.931,E2 28453.931} C_VEL
LIN {X 0,Y 600.09,Z 1080.384,A -85,B 0,C 180,E1 28453.048,E2 28453.048} C_VEL
LIN {X 0,Y 600.039,Z 1094.932,A -85,B 0,C 180,E1 28452.004,E2 28452.004} C_VEL
LIN {X 0,Y 600.001,Z 1108.524,A -85,B 0,C 180,E1 28450.806,E2 28450.806} C_VEL
LIN {X 0,Y 599.969,Z 1120.639,A -85,B 0,C 180,E1 28449.497,E2 28449.497} C_VEL
LIN {X 0,Y 599.949,Z 1130.906,A -85,B 0,C 180,E1 28448.131,E2 28448.131} C_VEL
LIN {X 0,Y 599.928,Z 1140.117,A -85,B 0,C 180,E1 28446.604,E2 28446.604} C_VEL
LIN {X 0,Y 599.921,Z 1147.351,A -85,B 0,C 180,E1 28445.068,E2 28445.068} C_VEL
LIN {X 0,Y 599.916,Z 1153.067,A -85,B 0,C 180,E1 28443.44,E2 28443.44} C_VEL
LIN {X 0,Y 599.914,Z 1156.896,A -85,B 0,C 180,E1 28441.815,E2 28441.815} C_VEL
LIN {X 0,Y 599.913,Z 1158.984,A -85,B 0,C 180,E1 28440.191,E2 28440.191} C_VEL
LIN {X 0,Y 599.913,Z 1159.396,A -85,B 0,C 180,E1 28438.472,E2 28438.472} C_VEL
LIN {X 0,Y 599.911,Z 1157.964,A -85,B 0,C 180,E1 28436.752,E2 28436.752} C_VEL
LIN {X 0,Y 599.918,Z 1154.817,A -85,B 0,C 180,E1 28435.124,E2 28435.124} C_VEL
LIN {X 0,Y 599.918,Z 1149.854,A -85,B 0,C 180,E1 28433.493,E2 28433.493} C_VEL
LIN {X 0,Y 599.923,Z 1142.928,A -85,B 0,C 180,E1 28431.856,E2 28431.856} C_VEL
LIN {X 0,Y 599.936,Z 1134.958,A -85,B 0,C 180,E1 28430.406,E2 28430.406} C_VEL
LIN {X 0,Y 599.961,Z 1124.943,A -85,B 0,C 180,E1 28428.951,E2 28428.951} C_VEL
LIN {X 0,Y 599.985,Z 1114.177,A -85,B 0,C 180,E1 28427.684,E2 28427.684} C_VEL
LIN {X 0,Y 600.021,Z 1101.005,A -85,B 0,C 180,E1 28426.411,E2 28426.411} C_VEL
LIN {X 0,Y 600.067,Z 1087.3,A -85,B 0,C 180,E1 28425.329,E2 28425.329} C_VEL
LIN {X 0,Y 600.109,Z 1072.215,A -85,B 0,C 180,E1 28424.371,E2 28424.371} C_VEL
LIN {X 0,Y 600.146,Z 1055.815,A -85,B 0,C 180,E1 28423.548,E2 28423.548} C_VEL
LIN {X 0,Y 600.189,Z 1038.787,A -85,B 0,C 180,E1 28422.901,E2 28422.901} C_VEL
LIN {X 0,Y 600.225,Z 1021.383,A -85,B 0,C 180,E1 28422.436,E2 28422.436} C_VEL
LIN {X 0,Y 600.246,Z 1001.344,A -85,B 0,C 180,E1 28422.124,E2 28422.124} C_VEL
LIN {X 0,Y 600.18,Z 844.669,A -85,B 0,C 180,E1 28420.183,E2 28420.183} C_VEL
LIN {X 0,Y 600.282,Z 800.81,A -85,B 0,C 180,E1 28417.01,E2 28417.01} C_VEL
LIN {X 0,Y 600.38,Z 758.995,A -85,B 0,C 180,E1 28413.918,E2 28413.918} C_VEL
LIN {X 0,Y 600.504,Z 719.275,A -85,B 0,C 180,E1 28410.91,E2 28410.91} C_VEL
LIN {X 0,Y 600.654,Z 679.506,A -85,B 0,C 180,E1 28407.814,E2 28407.814} C_VEL
LIN {X 0,Y 600.667,Z 662.443,A -85,B 0,C 180,E1 28406.452,E2 28406.452} C_VEL
LIN {X 0,Y 599.971,Z 660.002,A -85,B 0,C 180,E1 28406.178,E2 28406.178} C_VEL
LIN {X 0,Y 599.98,Z 660.003,A -85,B 0,C 180,E1 28402.896,E2 28402.896} C_VEL
LIN {X 0,Y 599.979,Z 660.105,A -85,B 0,C 180,E1 28399.774,E2 28399.774} C_VEL
LIN {X 0,Y 600.589,Z 663.422,A -85,B 0,C 180,E1 28399.576,E2 28399.576} C_VEL
LIN {X 0,Y 600.66,Z 734.815,A -85,B 0,C 180,E1 28396.394,E2 28396.394} C_VEL
LIN {X 0,Y 601.494,Z 747.669,A -85,B 0,C 180,E1 28395.721,E2 28395.721} C_VEL
LIN {X 0,Y 602.484,Z 756.908,A -85,B 0,C 180,E1 28395.078,E2 28395.078} C_VEL
LIN {X 0,Y 603.565,Z 763.359,A -85,B 0,C 180,E1 28394.44,E2 28394.44} C_VEL
LIN {X 0,Y 604.494,Z 766.811,A -85,B 0,C 180,E1 28393.872,E2 28393.872} C_VEL
LIN {X 0,Y 605.162,Z 767.998,A -85,B 0,C 180,E1 28393.367,E2 28393.367} C_VEL
LIN {X 0,Y 605.478,Z 767.375,A -85,B 0,C 180,E1 28392.872,E2 28392.872} C_VEL
LIN {X 0,Y 605.328,Z 765.089,A -85,B 0,C 180,E1 28392.451,E2 28392.451} C_VEL
LIN {X 0,Y 604.754,Z 761.159,A -85,B 0,C 180,E1 28392.103,E2 28392.103} C_VEL
LIN {X 0,Y 603.865,Z 755.128,A -85,B 0,C 180,E1 28391.849,E2 28391.849} C_VEL
LIN {X 0,Y 602.844,Z 746.004,A -85,B 0,C 180,E1 28391.715,E2 28391.715} C_VEL
LIN {X 0,Y 602.569,Z 737.506,A -85,B 0,C 180,E1 28391.686,E2 28391.686} C_VEL
LIN {X 0,Y 602.542,Z 664.957,A -85,B 0,C 180,E1 28391.683,E2 28391.683} C_VEL
LIN {X 0,Y 600.552,Z 662.187,A -85,B 0,C 180,E1 28391.469,E2 28391.469} C_VEL
LIN {X 0,Y 599.959,Z 660.004,A -85,B 0,C 180,E1 28391.389,E2 28391.389} C_VEL
LIN {X 0,Y 599.988,Z 660.111,A -85,B 0,C 180,E1 28388.649,E2 28388.649} C_VEL
LIN {X 0,Y 601.24,Z 663.666,A -85,B 0,C 180,E1 28388.338,E2 28388.338} C_VEL
LIN {X 0,Y 601.043,Z 713.363,A -85,B 0,C 180,E1 28385.4,E2 28385.4} C_VEL
LIN {X 0,Y 601.024,Z 759.54,A -85,B 0,C 180,E1 28382.782,E2 28382.782} C_VEL
LIN {X 0,Y 600.968,Z 937.788,A -85,B 0,C 180,E1 28380.337,E2 28380.337} C_VEL
LIN {X 0,Y 600.85,Z 1065.232,A -85,B 0,C 180,E1 28378.601,E2 28378.601} C_VEL
LIN {X 0,Y 600.794,Z 1086.514,A -85,B 0,C 180,E1 28378.131,E2 28378.131} C_VEL
LIN {X 0,Y 600.71,Z 1107.304,A -85,B 0,C 180,E1 28377.509,E2 28377.509} C_VEL
LIN {X 0,Y 600.63,Z 1128.56,A -85,B 0,C 180,E1 28376.68,E2 28376.68} C_VEL
LIN {X 0,Y 600.538,Z 1148.74,A -85,B 0,C 180,E1 28375.704,E2 28375.704} C_VEL
LIN {X 0,Y 600.435,Z 1167.924,A -85,B 0,C 180,E1 28374.602,E2 28374.602} C_VEL
LIN {X 0,Y 600.348,Z 1187.012,A -85,B 0,C 180,E1 28373.3,E2 28373.3} C_VEL
LIN {X 0,Y 600.247,Z 1204.55,A -85,B 0,C 180,E1 28371.903,E2 28371.903} C_VEL
LIN {X 0,Y 600.161,Z 1222.165,A -85,B 0,C 180,E1 28370.275,E2 28370.275} C_VEL
LIN {X 0,Y 600.091,Z 1237.317,A -85,B 0,C 180,E1 28368.658,E2 28368.658} C_VEL
LIN {X 0,Y 600.039,Z 1251.882,A -85,B 0,C 180,E1 28366.855,E2 28366.855} C_VEL
LIN {X 0,Y 599.993,Z 1264.18,A -85,B 0,C 180,E1 28365.068,E2 28365.068} C_VEL
LIN {X 0,Y 599.962,Z 1275.769,A -85,B 0,C 180,E1 28363.1,E2 28363.1} C_VEL
LIN {X 0,Y 599.938,Z 1285.423,A -85,B 0,C 180,E1 28361.147,E2 28361.147} C_VEL
LIN {X 0,Y 599.921,Z 1293.174,A -85,B 0,C 180,E1 28359.207,E2 28359.207} C_VEL
LIN {X 0,Y 599.909,Z 1299.888,A -85,B 0,C 180,E1 28357.085,E2 28357.085} C_VEL
LIN {X 0,Y 599.904,Z 1304.631,A -85,B 0,C 180,E1 28355.068,E2 28355.068} C_VEL
LIN {X 0,Y 599.907,Z 1307.674,A -85,B 0,C 180,E1 28353.058,E2 28353.058} C_VEL
LIN {X 0,Y 599.908,Z 1309.284,A -85,B 0,C 180,E1 28350.955,E2 28350.955} C_VEL
LIN {X 0,Y 599.913,Z 1309.262,A -85,B 0,C 180,E1 28348.95,E2 28348.95} C_VEL
LIN {X 0,Y 599.913,Z 1307.562,A -85,B 0,C 180,E1 28346.848,E2 28346.848} C_VEL
LIN {X 0,Y 599.911,Z 1304.223,A -85,B 0,C 180,E1 28344.741,E2 28344.741} C_VEL
LIN {X 0,Y 599.909,Z 1299.636,A -85,B 0,C 180,E1 28342.82,E2 28342.82} C_VEL
LIN {X 0,Y 599.921,Z 1293.178,A -85,B 0,C 180,E1 28340.794,E2 28340.794} C_VEL
LIN {X 0,Y 599.938,Z 1285.428,A -85,B 0,C 180,E1 28338.854,E2 28338.854} C_VEL
LIN {X 0,Y 599.962,Z 1275.773,A -85,B 0,C 180,E1 28336.901,E2 28336.901} C_VEL
LIN {X 0,Y 599.993,Z 1264.187,A -85,B 0,C 180,E1 28334.932,E2 28334.932} C_VEL
LIN {X 0,Y 600.038,Z 1251.887,A -85,B 0,C 180,E1 28333.146,E2 28333.146} C_VEL
LIN {X 0,Y 600.091,Z 1237.324,A -85,B 0,C 180,E1 28331.343,E2 28331.343} C_VEL
LIN {X 0,Y 600.161,Z 1222.009,A -85,B 0,C 180,E1 28329.709,E2 28329.709} C_VEL
LIN {X 0,Y 600.247,Z 1204.494,A -85,B 0,C 180,E1 28328.092,E2 28328.092} C_VEL
LIN {X 0,Y 600.348,Z 1187.024,A -85,B 0,C 180,E1 28326.7,E2 28326.7} C_VEL
LIN {X 0,Y 600.436,Z 1167.889,A -85,B 0,C 180,E1 28325.396,E2 28325.396} C_VEL
LIN {X 0,Y 600.538,Z 1148.758,A -85,B 0,C 180,E1 28324.297,E2 28324.297} C_VEL
LIN {X 0,Y 600.629,Z 1128.583,A -85,B 0,C 180,E1 28323.321,E2 28323.321} C_VEL
LIN {X 0,Y 600.709,Z 1107.476,A -85,B 0,C 180,E1 28322.497,E2 28322.497} C_VEL
LIN {X 0,Y 600.794,Z 1086.19,A -85,B 0,C 180,E1 28321.86,E2 28321.86} C_VEL
LIN {X 0,Y 600.85,Z 1064.757,A -85,B 0,C 180,E1 28321.391,E2 28321.391} C_VEL
LIN {X 0,Y 601.073,Z 825.892,A -85,B 0,C 180,E1 28318.14,E2 28318.14} C_VEL
LIN {X 0,Y 600.948,Z 759.095,A -85,B 0,C 180,E1 28317.207,E2 28317.207} C_VEL
LIN {X 0,Y 601.092,Z 704.808,A -85,B 0,C 180,E1 28314.103,E2 28314.103} C_VEL
LIN {X 0,Y 601.115,Z 663.242,A -85,B 0,C 180,E1 28311.627,E2 28311.627} C_VEL
LIN {X 0,Y 599.974,Z 660.004,A -85,B 0,C 180,E1 28311.323,E2 28311.323} C_VEL
LIN {X 0,Y 599.984,Z 660.194,A -85,B 0,C 180,E1 28308.592,E2 28308.592} C_VEL
LIN {X 0,Y 601.125,Z 663.277,A -85,B 0,C 180,E1 28308.469,E2 28308.469} C_VEL
LIN {X 0,Y 602.563,Z 664.975,A -85,B 0,C 180,E1 28308.315,E2 28308.315} C_VEL
LIN {X 0,Y 602.75,Z 744.421,A -85,B 0,C 180,E1 28308.295,E2 28308.295} C_VEL
LIN {X 0,Y 603.738,Z 754.221,A -85,B 0,C 180,E1 28308.174,E2 28308.174} C_VEL
LIN {X 0,Y 604.639,Z 760.353,A -85,B 0,C 180,E1 28307.943,E2 28307.943} C_VEL
LIN {X 0,Y 605.261,Z 764.605,A -85,B 0,C 180,E1 28307.609,E2 28307.609} C_VEL
LIN {X 0,Y 605.483,Z 767.167,A -85,B 0,C 180,E1 28307.188,E2 28307.188} C_VEL
LIN {X 0,Y 605.243,Z 768.033,A -85,B 0,C 180,E1 28306.72,E2 28306.72} C_VEL
LIN {X 0,Y 604.702,Z 767.31,A -85,B 0,C 180,E1 28306.267,E2 28306.267} C_VEL
LIN {X 0,Y 603.856,Z 764.667,A -85,B 0,C 180,E1 28305.735,E2 28305.735} C_VEL
LIN {X 0,Y 602.776,Z 758.931,A -85,B 0,C 180,E1 28305.096,E2 28305.096} C_VEL
LIN {X 0,Y 601.736,Z 749.613,A -85,B 0,C 180,E1 28304.39,E2 28304.39} C_VEL
LIN {X 0,Y 601.693,Z 695.621,A -85,B 0,C 180,E1 28300.88,E2 28300.88} C_VEL
LIN {X 0,Y 601.805,Z 664.202,A -85,B 0,C 180,E1 28298.721,E2 28298.721} C_VEL
LIN {X 0,Y 600.108,Z 660.783,A -85,B 0,C 180,E1 28298.301,E2 28298.301} C_VEL
LIN {X 0,Y 599.977,Z 660.003,A -85,B 0,C 180,E1 28298.19,E2 28298.19} C_VEL
LIN {X 0,Y 599.972,Z 660.004,A -85,B 0,C 180,E1 28294.924,E2 28294.924} C_VEL
LIN {X 0,Y 599.969,Z 660.001,A -85,B 0,C 180,E1 28291.665,E2 28291.665} C_VEL
LIN {X 0,Y 599.964,Z 660,A -85,B 0,C 180,E1 28288.357,E2 28288.357} C_VEL
LIN {X 0,Y 599.965,Z 659.999,A -85,B 0,C 180,E1 28285.148,E2 28285.148} C_VEL
LIN {X 0,Y 599.969,Z 659.998,A -85,B 0,C 180,E1 28281.919,E2 28281.919} C_VEL
LIN {X 0,Y 599.965,Z 659.999,A -85,B 0,C 180,E1 28278.661,E2 28278.661} C_VEL
LIN {X 0,Y 599.973,Z 660,A -85,B 0,C 180,E1 28275.365,E2 28275.365} C_VEL
LIN {X 0,Y 599.964,Z 660.003,A -85,B 0,C 180,E1 28272.121,E2 28272.121} C_VEL
LIN {X 0,Y 599.975,Z 660.004,A -85,B 0,C 180,E1 28268.916,E2 28268.916} C_VEL
LIN {X 0,Y 599.973,Z 660.004,A -85,B 0,C 180,E1 28265.738,E2 28265.738} C_VEL
LIN {X 0,Y 599.965,Z 660.003,A -85,B 0,C 180,E1 28262.483,E2 28262.483} C_VEL
LIN {X 0,Y 599.963,Z 660.001,A -85,B 0,C 180,E1 28259.236,E2 28259.236} C_VEL
LIN {X 0,Y 599.962,Z 660,A -85,B 0,C 180,E1 28255.986,E2 28255.986} C_VEL
LIN {X 0,Y 599.972,Z 660.004,A -85,B 0,C 180,E1 28253.437,E2 28253.437} C_VEL
LIN {X 0,Y 598.959,Z 660.133,A -85,B 0,C 180,E1 28252.702,E2 28252.702} C_VEL
LIN {X 0,Y 592.563,Z 660.929,A -85,B 0,C 180,E1 28250.638,E2 28250.638} C_VEL
LIN {X 0,Y 592.035,Z 660.99,A -85,B 0,C 180,E1 28250.101,E2 28250.101} C_VEL
LIN {X 0,Y 592.021,Z 660.989,A -85,B 0,C 180,E1 28246.82,E2 28246.82} C_VEL
LIN {X 0,Y 592.026,Z 660.988,A -85,B 0,C 180,E1 28243.591,E2 28243.591} C_VEL
LIN {X 0,Y 592.022,Z 660.987,A -85,B 0,C 180,E1 28240.361,E2 28240.361} C_VEL
LIN {X 0,Y 592.02,Z 660.988,A -85,B 0,C 180,E1 28237.142,E2 28237.142} C_VEL
LIN {X 0,Y 592.019,Z 660.989,A -85,B 0,C 180,E1 28233.952,E2 28233.952} C_VEL
LIN {X 0,Y 592.017,Z 660.984,A -85,B 0,C 180,E1 28230.784,E2 28230.784} C_VEL
LIN {X 0,Y 592.021,Z 660.99,A -85,B 0,C 180,E1 28227.611,E2 28227.611} C_VEL
LIN {X 0,Y 592.016,Z 660.987,A -85,B 0,C 180,E1 28224.48,E2 28224.48} C_VEL
LIN {X 0,Y 592.033,Z 660.991,A -85,B 0,C 180,E1 28221.282,E2 28221.282} C_VEL
LIN {X 0,Y 592.032,Z 660.991,A -85,B 0,C 180,E1 28217.995,E2 28217.995} C_VEL
LIN {X 0,Y 592.027,Z 660.994,A -85,B 0,C 180,E1 28214.769,E2 28214.769} C_VEL
LIN {X 0,Y 592.03,Z 660.993,A -85,B 0,C 180,E1 28211.568,E2 28211.568} C_VEL
LIN {X 0,Y 592.018,Z 660.993,A -85,B 0,C 180,E1 28208.404,E2 28208.404} C_VEL
LIN {X 0,Y 592.021,Z 661.006,A -85,B 0,C 180,E1 28205.216,E2 28205.216} C_VEL
LIN {X 0,Y 593.976,Z 667.078,A -85,B 0,C 180,E1 28204.677,E2 28204.677} C_VEL
LIN {X 0,Y 593.644,Z 713.746,A -85,B 0,C 180,E1 28201.644,E2 28201.644} C_VEL
LIN {X 0,Y 593.336,Z 763.058,A -85,B 0,C 180,E1 28198.537,E2 28198.537} C_VEL
LIN {X 0,Y 593.442,Z 766.285,A -85,B 0,C 180,E1 28198.369,E2 28198.369} C_VEL
LIN {X 0,Y 593.731,Z 772.82,A -85,B 0,C 180,E1 28198.266,E2 28198.266} C_VEL
LIN {X 0,Y 593.37,Z 1008.678,A -85,B 0,C 180,E1 28195.152,E2 28195.152} C_VEL
LIN {X 0,Y 593.308,Z 1033.466,A -85,B 0,C 180,E1 28194.766,E2 28194.766} C_VEL
LIN {X 0,Y 593.195,Z 1053.694,A -85,B 0,C 180,E1 28194.271,E2 28194.271} C_VEL
LIN {X 0,Y 593.069,Z 1073.583,A -85,B 0,C 180,E1 28193.603,E2 28193.603} C_VEL
LIN {X 0,Y 592.913,Z 1093.872,A -85,B 0,C 180,E1 28192.715,E2 28192.715} C_VEL
LIN {X 0,Y 592.758,Z 1112.92,A -85,B 0,C 180,E1 28191.678,E2 28191.678} C_VEL
LIN {X 0,Y 592.592,Z 1130.32,A -85,B 0,C 180,E1 28190.539,E2 28190.539} C_VEL
LIN {X 0,Y 592.428,Z 1148.005,A -85,B 0,C 180,E1 28189.163,E2 28189.163} C_VEL
LIN {X 0,Y 592.29,Z 1164.301,A -85,B 0,C 180,E1 28187.66,E2 28187.66} C_VEL
LIN {X 0,Y 592.172,Z 1178.88,A -85,B 0,C 180,E1 28186.075,E2 28186.075} C_VEL
LIN {X 0,Y 592.075,Z 1192.165,A -85,B 0,C 180,E1 28184.373,E2 28184.373} C_VEL
LIN {X 0,Y 592.012,Z 1203.347,A -85,B 0,C 180,E1 28182.683,E2 28182.683} C_VEL
LIN {X 0,Y 591.975,Z 1213.689,A -85,B 0,C 180,E1 28180.805,E2 28180.805} C_VEL
LIN {X 0,Y 591.933,Z 1222.005,A -85,B 0,C 180,E1 28178.94,E2 28178.94} C_VEL
LIN {X 0,Y 591.91,Z 1228.566,A -85,B 0,C 180,E1 28177.083,E2 28177.083} C_VEL
LIN {X 0,Y 591.906,Z 1233.754,A -85,B 0,C 180,E1 28175.136,E2 28175.136} C_VEL
LIN {X 0,Y 591.914,Z 1237.279,A -85,B 0,C 180,E1 28173.195,E2 28173.195} C_VEL
LIN {X 0,Y 591.912,Z 1239.175,A -85,B 0,C 180,E1 28171.161,E2 28171.161} C_VEL
LIN {X 0,Y 591.905,Z 1239.339,A -85,B 0,C 180,E1 28169.225,E2 28169.225} C_VEL
LIN {X 0,Y 591.909,Z 1237.943,A -85,B 0,C 180,E1 28167.289,E2 28167.289} C_VEL
LIN {X 0,Y 591.918,Z 1234.841,A -85,B 0,C 180,E1 28165.289,E2 28165.289} C_VEL
LIN {X 0,Y 591.927,Z 1230.118,A -85,B 0,C 180,E1 28163.328,E2 28163.328} C_VEL
LIN {X 0,Y 591.935,Z 1223.513,A -85,B 0,C 180,E1 28161.353,E2 28161.353} C_VEL
LIN {X 0,Y 591.963,Z 1215.504,A -85,B 0,C 180,E1 28159.489,E2 28159.489} C_VEL
LIN {X 0,Y 592,Z 1205.598,A -85,B 0,C 180,E1 28157.614,E2 28157.614} C_VEL
LIN {X 0,Y 592.074,Z 1194.207,A -85,B 0,C 180,E1 28155.826,E2 28155.826} C_VEL
LIN {X 0,Y 592.161,Z 1181.329,A -85,B 0,C 180,E1 28154.125,E2 28154.125} C_VEL
LIN {X 0,Y 592.279,Z 1166.92,A -85,B 0,C 180,E1 28152.513,E2 28152.513} C_VEL
LIN {X 0,Y 592.412,Z 1151.459,A -85,B 0,C 180,E1 28151.04,E2 28151.04} C_VEL
LIN {X 0,Y 592.567,Z 1134.377,A -85,B 0,C 180,E1 28149.66,E2 28149.66} C_VEL
LIN {X 0,Y 592.726,Z 1116.12,A -85,B 0,C 180,E1 28148.423,E2 28148.423} C_VEL
LIN {X 0,Y 592.862,Z 1097.648,A -85,B 0,C 180,E1 28147.386,E2 28147.386} C_VEL
LIN {X 0,Y 593.02,Z 1078.841,A -85,B 0,C 180,E1 28146.522,E2 28146.522} C_VEL
LIN {X 0,Y 593.182,Z 1058.49,A -85,B 0,C 180,E1 28145.785,E2 28145.785} C_VEL
LIN {X 0,Y 593.289,Z 1038.104,A -85,B 0,C 180,E1 28145.239,E2 28145.239} C_VEL
LIN {X 0,Y 593.358,Z 1017.109,A -85,B 0,C 180,E1 28144.868,E2 28144.868} C_VEL
LIN {X 0,Y 593.719,Z 781.309,A -85,B 0,C 180,E1 28141.758,E2 28141.758} C_VEL
LIN {X 0,Y 593.512,Z 769.713,A -85,B 0,C 180,E1 28141.591,E2 28141.591} C_VEL
LIN {X 0,Y 593.037,Z 767.211,A -85,B 0,C 180,E1 28141.501,E2 28141.501} C_VEL
LIN {X 0,Y 593.296,Z 730.591,A -85,B 0,C 180,E1 28138.221,E2 28138.221} C_VEL
LIN {X 0,Y 593.573,Z 695.769,A -85,B 0,C 180,E1 28134.995,E2 28134.995} C_VEL
LIN {X 0,Y 593.784,Z 666.283,A -85,B 0,C 180,E1 28132.161,E2 28132.161} C_VEL
LIN {X 0,Y 592.03,Z 660.99,A -85,B 0,C 180,E1 28131.512,E2 28131.512} C_VEL
LIN {X 0,Y 592.021,Z 660.991,A -85,B 0,C 180,E1 28128.285,E2 28128.285} C_VEL
LIN {X 0,Y 592.02,Z 660.985,A -85,B 0,C 180,E1 28125.044,E2 28125.044} C_VEL
LIN {X 0,Y 592.034,Z 660.992,A -85,B 0,C 180,E1 28121.844,E2 28121.844} C_VEL
LIN {X 0,Y 592.017,Z 660.986,A -85,B 0,C 180,E1 28118.675,E2 28118.675} C_VEL
LIN {X 0,Y 592.016,Z 660.992,A -85,B 0,C 180,E1 28115.506,E2 28115.506} C_VEL
LIN {X 0,Y 592.017,Z 660.991,A -85,B 0,C 180,E1 28112.37,E2 28112.37} C_VEL
LIN {X 0,Y 592.045,Z 661.162,A -85,B 0,C 180,E1 28112.097,E2 28112.097} C_VEL
LIN {X 0,Y 593.501,Z 666.154,A -85,B 0,C 180,E1 28111.597,E2 28111.597} C_VEL
LIN {X 0,Y 593.233,Z 704.331,A -85,B 0,C 180,E1 28108.549,E2 28108.549} C_VEL
LIN {X 0,Y 592.971,Z 744.783,A -85,B 0,C 180,E1 28105.413,E2 28105.413} C_VEL
LIN {X 0,Y 592.748,Z 785.912,A -85,B 0,C 180,E1 28102.305,E2 28102.305} C_VEL
LIN {X 0,Y 592.539,Z 830.579,A -85,B 0,C 180,E1 28099.006,E2 28099.006} C_VEL
LIN {X 0,Y 592.522,Z 845.225,A -85,B 0,C 180,E1 28097.962,E2 28097.962} C_VEL
LIN {X 0,Y 592.565,Z 1011.553,A -85,B 0,C 180,E1 28095.873,E2 28095.873} C_VEL
LIN {X 0,Y 592.52,Z 1028.426,A -85,B 0,C 180,E1 28095.525,E2 28095.525} C_VEL
LIN {X 0,Y 592.461,Z 1044.91,A -85,B 0,C 180,E1 28095.014,E2 28095.014} C_VEL
LIN {X 0,Y 592.361,Z 1061.55,A -85,B 0,C 180,E1 28094.302,E2 28094.302} C_VEL
LIN {X 0,Y 592.268,Z 1077.438,A -85,B 0,C 180,E1 28093.422,E2 28093.422} C_VEL
LIN {X 0,Y 592.192,Z 1092.408,A -85,B 0,C 180,E1 28092.382,E2 28092.382} C_VEL
LIN {X 0,Y 592.104,Z 1106.157,A -85,B 0,C 180,E1 28091.198,E2 28091.198} C_VEL
LIN {X 0,Y 592.034,Z 1119.107,A -85,B 0,C 180,E1 28089.821,E2 28089.821} C_VEL
LIN {X 0,Y 591.987,Z 1129.593,A -85,B 0,C 180,E1 28088.45,E2 28088.45} C_VEL
LIN {X 0,Y 591.951,Z 1138.65,A -85,B 0,C 180,E1 28086.985,E2 28086.985} C_VEL
LIN {X 0,Y 591.927,Z 1146.198,A -85,B 0,C 180,E1 28085.428,E2 28085.428} C_VEL
LIN {X 0,Y 591.921,Z 1152.206,A -85,B 0,C 180,E1 28083.777,E2 28083.777} C_VEL
LIN {X 0,Y 591.915,Z 1156.37,A -85,B 0,C 180,E1 28082.13,E2 28082.13} C_VEL
LIN {X 0,Y 591.916,Z 1158.776,A -85,B 0,C 180,E1 28080.484,E2 28080.484} C_VEL
LIN {X 0,Y 591.914,Z 1159.482,A -85,B 0,C 180,E1 28078.839,E2 28078.839} C_VEL
LIN {X 0,Y 591.916,Z 1158.406,A -85,B 0,C 180,E1 28077.095,E2 28077.095} C_VEL
LIN {X 0,Y 591.914,Z 1155.464,A -85,B 0,C 180,E1 28075.349,E2 28075.349} C_VEL
LIN {X 0,Y 591.919,Z 1150.844,A -85,B 0,C 180,E1 28073.697,E2 28073.697} C_VEL
LIN {X 0,Y 591.934,Z 1144.243,A -85,B 0,C 180,E1 28072.039,E2 28072.039} C_VEL
LIN {X 0,Y 591.958,Z 1136.024,A -85,B 0,C 180,E1 28070.472,E2 28070.472} C_VEL
LIN {X 0,Y 592,Z 1126.296,A -85,B 0,C 180,E1 28068.998,E2 28068.998} C_VEL
LIN {X 0,Y 592.056,Z 1114.958,A -85,B 0,C 180,E1 28067.615,E2 28067.615} C_VEL
LIN {X 0,Y 592.124,Z 1102.505,A -85,B 0,C 180,E1 28066.376,E2 28066.376} C_VEL
LIN {X 0,Y 592.219,Z 1087.785,A -85,B 0,C 180,E1 28065.18,E2 28065.18} C_VEL
LIN {X 0,Y 592.307,Z 1072.622,A -85,B 0,C 180,E1 28064.197,E2 28064.197} C_VEL
LIN {X 0,Y 592.39,Z 1056.618,A -85,B 0,C 180,E1 28063.376,E2 28063.376} C_VEL
LIN {X 0,Y 592.471,Z 1039.838,A -85,B 0,C 180,E1 28062.722,E2 28062.722} C_VEL
LIN {X 0,Y 592.532,Z 1023.017,A -85,B 0,C 180,E1 28062.255,E2 28062.255} C_VEL
LIN {X 0,Y 592.584,Z 1004.98,A -85,B 0,C 180,E1 28061.945,E2 28061.945} C_VEL
LIN {X 0,Y 592.538,Z 845.36,A -85,B 0,C 180,E1 28059.95,E2 28059.95} C_VEL
LIN {X 0,Y 592.597,Z 815.449,A -85,B 0,C 180,E1 28057.794,E2 28057.794} C_VEL
LIN {X 0,Y 592.809,Z 772.957,A -85,B 0,C 180,E1 28054.634,E2 28054.634} C_VEL
LIN {X 0,Y 593.067,Z 731.086,A -85,B 0,C 180,E1 28051.445,E2 28051.445} C_VEL
LIN {X 0,Y 593.311,Z 692.075,A -85,B 0,C 180,E1 28048.392,E2 28048.392} C_VEL
LIN {X 0,Y 593.522,Z 665.85,A -85,B 0,C 180,E1 28046.29,E2 28046.29} C_VEL
LIN {X 0,Y 592.522,Z 662.927,A -85,B 0,C 180,E1 28045.95,E2 28045.95} C_VEL
LIN {X 0,Y 592.033,Z 660.995,A -85,B 0,C 180,E1 28045.504,E2 28045.504} C_VEL
LIN {X 0,Y 592.015,Z 660.993,A -85,B 0,C 180,E1 28042.311,E2 28042.311} C_VEL
LIN {X 0,Y 592.072,Z 661.237,A -85,B 0,C 180,E1 28040.332,E2 28040.332} C_VEL
LIN {X 0,Y 593.695,Z 665.366,A -85,B 0,C 180,E1 28039.919,E2 28039.919} C_VEL
LIN {X 0,Y 592.931,Z 692.817,A -85,B 0,C 180,E1 28038.59,E2 28038.59} C_VEL
LIN {X 0,Y 593.184,Z 738.061,A -85,B 0,C 180,E1 28036.517,E2 28036.517} C_VEL
LIN {X 0,Y 594.785,Z 754.566,A -85,B 0,C 180,E1 28035.696,E2 28035.696} C_VEL
LIN {X 0,Y 596.673,Z 763.635,A -85,B 0,C 180,E1 28035.132,E2 28035.132} C_VEL
LIN {X 0,Y 598.455,Z 769.344,A -85,B 0,C 180,E1 28034.624,E2 28034.624} C_VEL
LIN {X 0,Y 600.181,Z 773.083,A -85,B 0,C 180,E1 28034.109,E2 28034.109} C_VEL
LIN {X 0,Y 601.698,Z 775.089,A -85,B 0,C 180,E1 28033.572,E2 28033.572} C_VEL
LIN {X 0,Y 602.611,Z 775.468,A -85,B 0,C 180,E1 28033.11,E2 28033.11} C_VEL
LIN {X 0,Y 603.063,Z 774.341,A -85,B 0,C 180,E1 28032.567,E2 28032.567} C_VEL
LIN {X 0,Y 602.709,Z 771.619,A -85,B 0,C 180,E1 28032.084,E2 28032.084} C_VEL
LIN {X 0,Y 601.645,Z 767.534,A -85,B 0,C 180,E1 28031.695,E2 28031.695} C_VEL
LIN {X 0,Y 600.008,Z 761.845,A -85,B 0,C 180,E1 28031.412,E2 28031.412} C_VEL
LIN {X 0,Y 598.24,Z 753.431,A -85,B 0,C 180,E1 28031.218,E2 28031.218} C_VEL
LIN {X 0,Y 597.346,Z 741.794,A -85,B 0,C 180,E1 28031.12,E2 28031.12} C_VEL
LIN {X 0,Y 597.171,Z 668.583,A -85,B 0,C 180,E1 28031.101,E2 28031.101} C_VEL
LIN {X 0,Y 596.104,Z 667.002,A -85,B 0,C 180,E1 28030.983,E2 28030.983} C_VEL
LIN {X 0,Y 593.407,Z 664.591,A -85,B 0,C 180,E1 28030.683,E2 28030.683} C_VEL
LIN {X 0,Y 592.106,Z 661.548,A -85,B 0,C 180,E1 28030.536,E2 28030.536} C_VEL
LIN {X 0,Y 592.017,Z 660.992,A -85,B 0,C 180,E1 28030.517,E2 28030.517} C_VEL
LIN {X 0,Y 592.028,Z 661.073,A -85,B 0,C 180,E1 28029.208,E2 28029.208} C_VEL
LIN {X 0,Y 593.408,Z 664.58,A -85,B 0,C 180,E1 28028.882,E2 28028.882} C_VEL
LIN {X 0,Y 594.589,Z 667.677,A -85,B 0,C 180,E1 28028.6,E2 28028.6} C_VEL
LIN {X 0,Y 594.198,Z 717.813,A -85,B 0,C 180,E1 28025.607,E2 28025.607} C_VEL
LIN {X 0,Y 594.033,Z 759.494,A -85,B 0,C 180,E1 28023.218,E2 28023.218} C_VEL
LIN {X 0,Y 594.407,Z 764.186,A -85,B 0,C 180,E1 28023.128,E2 28023.128} C_VEL
LIN {X 0,Y 593.961,Z 998.242,A -85,B 0,C 180,E1 28019.904,E2 28019.904} C_VEL
LIN {X 0,Y 593.812,Z 1066.141,A -85,B 0,C 180,E1 28018.957,E2 28018.957} C_VEL
LIN {X 0,Y 593.696,Z 1087.814,A -85,B 0,C 180,E1 28018.464,E2 28018.464} C_VEL
LIN {X 0,Y 593.517,Z 1110.251,A -85,B 0,C 180,E1 28017.762,E2 28017.762} C_VEL
LIN {X 0,Y 593.343,Z 1131.563,A -85,B 0,C 180,E1 28016.902,E2 28016.902} C_VEL
LIN {X 0,Y 593.163,Z 1151.73,A -85,B 0,C 180,E1 28015.886,E2 28015.886} C_VEL
LIN {X 0,Y 592.944,Z 1171.139,A -85,B 0,C 180,E1 28014.721,E2 28014.721} C_VEL
LIN {X 0,Y 592.763,Z 1189.593,A -85,B 0,C 180,E1 28013.422,E2 28013.422} C_VEL
LIN {X 0,Y 592.583,Z 1208.098,A -85,B 0,C 180,E1 28011.894,E2 28011.894} C_VEL
LIN {X 0,Y 592.406,Z 1224.696,A -85,B 0,C 180,E1 28010.295,E2 28010.295} C_VEL
LIN {X 0,Y 592.26,Z 1239.871,A -85,B 0,C 180,E1 28008.607,E2 28008.607} C_VEL
LIN {X 0,Y 592.138,Z 1254.041,A -85,B 0,C 180,E1 28006.783,E2 28006.783} C_VEL
LIN {X 0,Y 592.054,Z 1266.743,A -85,B 0,C 180,E1 28004.875,E2 28004.875} C_VEL
LIN {X 0,Y 591.999,Z 1277.435,A -85,B 0,C 180,E1 28002.961,E2 28002.961} C_VEL
LIN {X 0,Y 591.954,Z 1287.07,A -85,B 0,C 180,E1 28000.905,E2 28000.905} C_VEL
LIN {X 0,Y 591.93,Z 1294.97,A -85,B 0,C 180,E1 27998.83,E2 27998.83} C_VEL
LIN {X 0,Y 591.919,Z 1300.905,A -85,B 0,C 180,E1 27996.791,E2 27996.791} C_VEL
LIN {X 0,Y 591.909,Z 1305.468,A -85,B 0,C 180,E1 27994.651,E2 27994.651} C_VEL
LIN {X 0,Y 591.901,Z 1308.33,A -85,B 0,C 180,E1 27992.518,E2 27992.518} C_VEL
LIN {X 0,Y 591.894,Z 1309.395,A -85,B 0,C 180,E1 27990.484,E2 27990.484} C_VEL
LIN {X 0,Y 591.895,Z 1308.885,A -85,B 0,C 180,E1 27988.258,E2 27988.258} C_VEL
LIN {X 0,Y 591.895,Z 1306.871,A -85,B 0,C 180,E1 27986.223,E2 27986.223} C_VEL
LIN {X 0,Y 591.908,Z 1303.195,A -85,B 0,C 180,E1 27984.183,E2 27984.183} C_VEL
LIN {X 0,Y 591.924,Z 1297.676,A -85,B 0,C 180,E1 27982.039,E2 27982.039} C_VEL
LIN {X 0,Y 591.946,Z 1291.052,A -85,B 0,C 180,E1 27980.08,E2 27980.08} C_VEL
LIN {X 0,Y 591.975,Z 1282.683,A -85,B 0,C 180,E1 27978.109,E2 27978.109} C_VEL
LIN {X 0,Y 592.022,Z 1272.55,A -85,B 0,C 180,E1 27976.124,E2 27976.124} C_VEL
LIN {X 0,Y 592.077,Z 1261.304,A -85,B 0,C 180,E1 27974.275,E2 27974.275} C_VEL
LIN {X 0,Y 592.183,Z 1248.02,A -85,B 0,C 180,E1 27972.409,E2 27972.409} C_VEL
LIN {X 0,Y 592.323,Z 1232.809,A -85,B 0,C 180,E1 27970.577,E2 27970.577} C_VEL
LIN {X 0,Y 592.487,Z 1217.016,A -85,B 0,C 180,E1 27968.934,E2 27968.934} C_VEL
LIN {X 0,Y 592.668,Z 1199.199,A -85,B 0,C 180,E1 27967.34,E2 27967.34} C_VEL
LIN {X 0,Y 592.829,Z 1181.212,A -85,B 0,C 180,E1 27965.965,E2 27965.965} C_VEL
LIN {X 0,Y 593.052,Z 1161.875,A -85,B 0,C 180,E1 27964.699,E2 27964.699} C_VEL
LIN {X 0,Y 593.259,Z 1142.748,A -85,B 0,C 180,E1 27963.635,E2 27963.635} C_VEL
LIN {X 0,Y 593.416,Z 1122.803,A -85,B 0,C 180,E1 27962.723,E2 27962.723} C_VEL
LIN {X 0,Y 593.599,Z 1101.086,A -85,B 0,C 180,E1 27961.927,E2 27961.927} C_VEL
LIN {X 0,Y 593.738,Z 1079.9,A -85,B 0,C 180,E1 27961.331,E2 27961.331} C_VEL
LIN {X 0,Y 593.831,Z 1058.449,A -85,B 0,C 180,E1 27960.919,E2 27960.919} C_VEL
LIN {X 0,Y 594.276,Z 825.256,A -85,B 0,C 180,E1 27957.723,E2 27957.723} C_VEL
LIN {X 0,Y 594.221,Z 760.553,A -85,B 0,C 180,E1 27956.808,E2 27956.808} C_VEL
LIN {X 0,Y 593.923,Z 757.94,A -85,B 0,C 180,E1 27956.715,E2 27956.715} C_VEL
LIN {X 0,Y 594.311,Z 704.795,A -85,B 0,C 180,E1 27953.628,E2 27953.628} C_VEL
LIN {X 0,Y 594.558,Z 667.265,A -85,B 0,C 180,E1 27951.373,E2 27951.373} C_VEL
LIN {X 0,Y 592.078,Z 661.393,A -85,B 0,C 180,E1 27950.816,E2 27950.816} C_VEL
LIN {X 0,Y 592.017,Z 660.993,A -85,B 0,C 180,E1 27950.767,E2 27950.767} C_VEL
LIN {X 0,Y 592.048,Z 661.219,A -85,B 0,C 180,E1 27949.471,E2 27949.471} C_VEL
LIN {X 0,Y 593.157,Z 664.214,A -85,B 0,C 180,E1 27949.346,E2 27949.346} C_VEL
LIN {X 0,Y 595.606,Z 666.704,A -85,B 0,C 180,E1 27949.072,E2 27949.072} C_VEL
LIN {X 0,Y 596.672,Z 667.693,A -85,B 0,C 180,E1 27948.954,E2 27948.954} C_VEL
LIN {X 0,Y 597.274,Z 668.977,A -85,B 0,C 180,E1 27948.888,E2 27948.888} C_VEL
LIN {X 0,Y 597.458,Z 744.734,A -85,B 0,C 180,E1 27948.868,E2 27948.868} C_VEL
LIN {X 0,Y 598.564,Z 755.532,A -85,B 0,C 180,E1 27948.747,E2 27948.747} C_VEL
LIN {X 0,Y 600.426,Z 763.322,A -85,B 0,C 180,E1 27948.534,E2 27948.534} C_VEL
LIN {X 0,Y 601.949,Z 768.602,A -85,B 0,C 180,E1 27948.223,E2 27948.223} C_VEL
LIN {X 0,Y 602.867,Z 772.453,A -85,B 0,C 180,E1 27947.803,E2 27947.803} C_VEL
LIN {X 0,Y 603.027,Z 774.771,A -85,B 0,C 180,E1 27947.302,E2 27947.302} C_VEL
LIN {X 0,Y 602.413,Z 775.497,A -85,B 0,C 180,E1 27946.772,E2 27946.772} C_VEL
LIN {X 0,Y 601.129,Z 774.484,A -85,B 0,C 180,E1 27946.209,E2 27946.209} C_VEL
LIN {X 0,Y 599.432,Z 771.672,A -85,B 0,C 180,E1 27945.662,E2 27945.662} C_VEL
LIN {X 0,Y 597.569,Z 766.742,A -85,B 0,C 180,E1 27945.121,E2 27945.121} C_VEL
LIN {X 0,Y 595.646,Z 757.059,A -85,B 0,C 180,E1 27944.351,E2 27944.351} C_VEL
LIN {X 0,Y 595.088,Z 741.764,A -85,B 0,C 180,E1 27943.322,E2 27943.322} C_VEL
LIN {X 0,Y 595.489,Z 700.069,A -85,B 0,C 180,E1 27940.589,E2 27940.589} C_VEL
LIN {X 0,Y 595.815,Z 669.073,A -85,B 0,C 180,E1 27938.444,E2 27938.444} C_VEL
LIN {X 0,Y 594.191,Z 665.536,A -85,B 0,C 180,E1 27938.015,E2 27938.015} C_VEL
LIN {X 0,Y 592.535,Z 662.983,A -85,B 0,C 180,E1 27937.651,E2 27937.651} C_VEL
LIN {X 0,Y 592.024,Z 660.991,A -85,B 0,C 180,E1 27937.445,E2 27937.445} C_VEL
LIN {X 0,Y 592.027,Z 660.99,A -85,B 0,C 180,E1 27934.154,E2 27934.154} C_VEL
LIN {X 0,Y 592.028,Z 660.99,A -85,B 0,C 180,E1 27930.891,E2 27930.891} C_VEL
LIN {X 0,Y 592.036,Z 660.991,A -85,B 0,C 180,E1 27927.547,E2 27927.547} C_VEL
LIN {X 0,Y 592.031,Z 660.993,A -85,B 0,C 180,E1 27924.335,E2 27924.335} C_VEL
LIN {X 0,Y 592.033,Z 660.992,A -85,B 0,C 180,E1 27921.083,E2 27921.083} C_VEL
LIN {X 0,Y 592.033,Z 660.989,A -85,B 0,C 180,E1 27917.73,E2 27917.73} C_VEL
LIN {X 0,Y 592.028,Z 660.988,A -85,B 0,C 180,E1 27914.375,E2 27914.375} C_VEL
LIN {X 0,Y 592.029,Z 660.988,A -85,B 0,C 180,E1 27911.1,E2 27911.1} C_VEL
LIN {X 0,Y 592.025,Z 660.988,A -85,B 0,C 180,E1 27907.862,E2 27907.862} C_VEL
LIN {X 0,Y 592.034,Z 660.989,A -85,B 0,C 180,E1 27904.552,E2 27904.552} C_VEL
LIN {X 0,Y 592.028,Z 660.993,A -85,B 0,C 180,E1 27901.258,E2 27901.258} C_VEL
LIN {X 0,Y 592.036,Z 660.992,A -85,B 0,C 180,E1 27898.064,E2 27898.064} C_VEL
LIN {X 0,Y 592.034,Z 660.992,A -85,B 0,C 180,E1 27894.864,E2 27894.864} C_VEL
LIN {X 0,Y 592.023,Z 660.991,A -85,B 0,C 180,E1 27891.648,E2 27891.648} C_VEL
LIN {X 0,Y 592.035,Z 660.99,A -85,B 0,C 180,E1 27890.101,E2 27890.101} C_VEL
LIN {X 0,Y 591.041,Z 661.112,A -85,B 0,C 180,E1 27889.355,E2 27889.355} C_VEL
LIN {X 0,Y 584.604,Z 661.918,A -85,B 0,C 180,E1 27887.264,E2 27887.264} C_VEL
LIN {X 0,Y 584.088,Z 661.977,A -85,B 0,C 180,E1 27886.719,E2 27886.719} C_VEL
LIN {X 0,Y 584.094,Z 661.976,A -85,B 0,C 180,E1 27883.389,E2 27883.389} C_VEL
LIN {X 0,Y 584.093,Z 661.976,A -85,B 0,C 180,E1 27879.979,E2 27879.979} C_VEL
LIN {X 0,Y 584.101,Z 661.977,A -85,B 0,C 180,E1 27876.707,E2 27876.707} C_VEL
LIN {X 0,Y 584.096,Z 661.979,A -85,B 0,C 180,E1 27873.353,E2 27873.353} C_VEL
LIN {X 0,Y 584.087,Z 661.979,A -85,B 0,C 180,E1 27870.123,E2 27870.123} C_VEL
LIN {X 0,Y 584.087,Z 661.978,A -85,B 0,C 180,E1 27866.902,E2 27866.902} C_VEL
LIN {X 0,Y 584.087,Z 661.976,A -85,B 0,C 180,E1 27863.68,E2 27863.68} C_VEL
LIN {X 0,Y 584.087,Z 661.975,A -85,B 0,C 180,E1 27860.446,E2 27860.446} C_VEL
LIN {X 0,Y 584.086,Z 661.977,A -85,B 0,C 180,E1 27857.187,E2 27857.187} C_VEL
LIN {X 0,Y 584.089,Z 661.978,A -85,B 0,C 180,E1 27854.026,E2 27854.026} C_VEL
LIN {X 0,Y 584.095,Z 661.98,A -85,B 0,C 180,E1 27850.682,E2 27850.682} C_VEL
LIN {X 0,Y 584.086,Z 661.982,A -85,B 0,C 180,E1 27847.411,E2 27847.411} C_VEL
LIN {X 0,Y 584.103,Z 662.032,A -85,B 0,C 180,E1 27845.697,E2 27845.697} C_VEL
LIN {X 0,Y 587.022,Z 670.085,A -85,B 0,C 180,E1 27844.946,E2 27844.946} C_VEL
LIN {X 0,Y 586.527,Z 716.399,A -85,B 0,C 180,E1 27841.901,E2 27841.901} C_VEL
LIN {X 0,Y 586.109,Z 765.794,A -85,B 0,C 180,E1 27838.764,E2 27838.764} C_VEL
LIN {X 0,Y 586.692,Z 771.299,A -85,B 0,C 180,E1 27838.658,E2 27838.658} C_VEL
LIN {X 0,Y 586.131,Z 1007.981,A -85,B 0,C 180,E1 27835.495,E2 27835.495} C_VEL
LIN {X 0,Y 586.033,Z 1033.34,A -85,B 0,C 180,E1 27835.098,E2 27835.098} C_VEL
LIN {X 0,Y 585.866,Z 1053.704,A -85,B 0,C 180,E1 27834.596,E2 27834.596} C_VEL
LIN {X 0,Y 585.682,Z 1073.597,A -85,B 0,C 180,E1 27833.919,E2 27833.919} C_VEL
LIN {X 0,Y 585.453,Z 1092.762,A -85,B 0,C 180,E1 27833.075,E2 27833.075} C_VEL
LIN {X 0,Y 585.213,Z 1111.155,A -85,B 0,C 180,E1 27832.078,E2 27832.078} C_VEL
LIN {X 0,Y 584.955,Z 1129.406,A -85,B 0,C 180,E1 27830.886,E2 27830.886} C_VEL
LIN {X 0,Y 584.718,Z 1146.749,A -85,B 0,C 180,E1 27829.535,E2 27829.535} C_VEL
LIN {X 0,Y 584.52,Z 1162.504,A -85,B 0,C 180,E1 27828.087,E2 27828.087} C_VEL
LIN {X 0,Y 584.343,Z 1177.191,A -85,B 0,C 180,E1 27826.501,E2 27826.501} C_VEL
LIN {X 0,Y 584.202,Z 1190.048,A -85,B 0,C 180,E1 27824.875,E2 27824.875} C_VEL
LIN {X 0,Y 584.093,Z 1202.144,A -85,B 0,C 180,E1 27823.059,E2 27823.059} C_VEL
LIN {X 0,Y 584.011,Z 1212.522,A -85,B 0,C 180,E1 27821.184,E2 27821.184} C_VEL
LIN {X 0,Y 583.951,Z 1221.196,A -85,B 0,C 180,E1 27819.262,E2 27819.262} C_VEL
LIN {X 0,Y 583.918,Z 1228.266,A -85,B 0,C 180,E1 27817.279,E2 27817.279} C_VEL
LIN {X 0,Y 583.917,Z 1233.345,A -85,B 0,C 180,E1 27815.404,E2 27815.404} C_VEL
LIN {X 0,Y 583.908,Z 1236.984,A -85,B 0,C 180,E1 27813.435,E2 27813.435} C_VEL
LIN {X 0,Y 583.901,Z 1238.976,A -85,B 0,C 180,E1 27811.471,E2 27811.471} C_VEL
LIN {X 0,Y 583.9,Z 1239.384,A -85,B 0,C 180,E1 27809.411,E2 27809.411} C_VEL
LIN {X 0,Y 583.908,Z 1238.054,A -85,B 0,C 180,E1 27807.35,E2 27807.35} C_VEL
LIN {X 0,Y 583.917,Z 1235.171,A -85,B 0,C 180,E1 27805.383,E2 27805.383} C_VEL
LIN {X 0,Y 583.93,Z 1230.591,A -85,B 0,C 180,E1 27803.412,E2 27803.412} C_VEL
LIN {X 0,Y 583.936,Z 1224.573,A -85,B 0,C 180,E1 27801.532,E2 27801.532} C_VEL
LIN {X 0,Y 583.982,Z 1216.426,A -85,B 0,C 180,E1 27799.543,E2 27799.543} C_VEL
LIN {X 0,Y 584.048,Z 1206.752,A -85,B 0,C 180,E1 27797.643,E2 27797.643} C_VEL
LIN {X 0,Y 584.152,Z 1195.606,A -85,B 0,C 180,E1 27795.832,E2 27795.832} C_VEL
LIN {X 0,Y 584.281,Z 1182.905,A -85,B 0,C 180,E1 27794.098,E2 27794.098} C_VEL
LIN {X 0,Y 584.463,Z 1167.911,A -85,B 0,C 180,E1 27792.374,E2 27792.374} C_VEL
LIN {X 0,Y 584.672,Z 1152.047,A -85,B 0,C 180,E1 27790.831,E2 27790.831} C_VEL
LIN {X 0,Y 584.901,Z 1135.047,A -85,B 0,C 180,E1 27789.433,E2 27789.433} C_VEL
LIN {X 0,Y 585.141,Z 1116.915,A -85,B 0,C 180,E1 27788.182,E2 27788.182} C_VEL
LIN {X 0,Y 585.357,Z 1098.634,A -85,B 0,C 180,E1 27787.132,E2 27787.132} C_VEL
LIN {X 0,Y 585.599,Z 1079.419,A -85,B 0,C 180,E1 27786.231,E2 27786.231} C_VEL
LIN {X 0,Y 585.837,Z 1059.024,A -85,B 0,C 180,E1 27785.479,E2 27785.479} C_VEL
LIN {X 0,Y 586.002,Z 1038.484,A -85,B 0,C 180,E1 27784.92,E2 27784.92} C_VEL
LIN {X 0,Y 586.109,Z 1017.595,A -85,B 0,C 180,E1 27784.542,E2 27784.542} C_VEL
LIN {X 0,Y 586.666,Z 781.767,A -85,B 0,C 180,E1 27781.394,E2 27781.394} C_VEL
LIN {X 0,Y 586.479,Z 771.344,A -85,B 0,C 180,E1 27781.242,E2 27781.242} C_VEL
LIN {X 0,Y 585.622,Z 767.482,A -85,B 0,C 180,E1 27781.132,E2 27781.132} C_VEL
LIN {X 0,Y 586.008,Z 731.825,A -85,B 0,C 180,E1 27777.894,E2 27777.894} C_VEL
LIN {X 0,Y 586.429,Z 697.685,A -85,B 0,C 180,E1 27774.69,E2 27774.69} C_VEL
LIN {X 0,Y 586.686,Z 669.663,A -85,B 0,C 180,E1 27771.986,E2 27771.986} C_VEL
LIN {X 0,Y 584.092,Z 661.977,A -85,B 0,C 180,E1 27771.08,E2 27771.08} C_VEL
LIN {X 0,Y 584.09,Z 661.982,A -85,B 0,C 180,E1 27767.836,E2 27767.836} C_VEL
LIN {X 0,Y 584.096,Z 661.974,A -85,B 0,C 180,E1 27764.575,E2 27764.575} C_VEL
LIN {X 0,Y 584.084,Z 661.974,A -85,B 0,C 180,E1 27761.228,E2 27761.228} C_VEL
LIN {X 0,Y 584.099,Z 661.981,A -85,B 0,C 180,E1 27757.918,E2 27757.918} C_VEL
LIN {X 0,Y 584.08,Z 661.977,A -85,B 0,C 180,E1 27754.634,E2 27754.634} C_VEL
LIN {X 0,Y 584.11,Z 662.182,A -85,B 0,C 180,E1 27752.543,E2 27752.543} C_VEL
LIN {X 0,Y 586.315,Z 669.15,A -85,B 0,C 180,E1 27751.8,E2 27751.8} C_VEL
LIN {X 0,Y 585.91,Z 708.092,A -85,B 0,C 180,E1 27748.655,E2 27748.655} C_VEL
LIN {X 0,Y 585.501,Z 748.478,A -85,B 0,C 180,E1 27745.489,E2 27745.489} C_VEL
LIN {X 0,Y 585.164,Z 788.912,A -85,B 0,C 180,E1 27742.398,E2 27742.398} C_VEL
LIN {X 0,Y 584.856,Z 832.184,A -85,B 0,C 180,E1 27739.162,E2 27739.162} C_VEL
LIN {X 0,Y 584.834,Z 845.317,A -85,B 0,C 180,E1 27738.22,E2 27738.22} C_VEL
LIN {X 0,Y 585.154,Z 853.436,A -85,B 0,C 180,E1 27738.106,E2 27738.106} C_VEL
LIN {X 0,Y 584.889,Z 1015.32,A -85,B 0,C 180,E1 27736.039,E2 27736.039} C_VEL
LIN {X 0,Y 584.812,Z 1033.792,A -85,B 0,C 180,E1 27735.599,E2 27735.599} C_VEL
LIN {X 0,Y 584.697,Z 1050.351,A -85,B 0,C 180,E1 27735.015,E2 27735.015} C_VEL
LIN {X 0,Y 584.56,Z 1066.493,A -85,B 0,C 180,E1 27734.259,E2 27734.259} C_VEL
LIN {X 0,Y 584.432,Z 1081.532,A -85,B 0,C 180,E1 27733.354,E2 27733.354} C_VEL
LIN {X 0,Y 584.303,Z 1095.056,A -85,B 0,C 180,E1 27732.351,E2 27732.351} C_VEL
LIN {X 0,Y 584.183,Z 1108.887,A -85,B 0,C 180,E1 27731.096,E2 27731.096} C_VEL
LIN {X 0,Y 584.085,Z 1120.855,A -85,B 0,C 180,E1 27729.757,E2 27729.757} C_VEL
LIN {X 0,Y 584.016,Z 1131.014,A -85,B 0,C 180,E1 27728.368,E2 27728.368} C_VEL
LIN {X 0,Y 583.961,Z 1140.79,A -85,B 0,C 180,E1 27726.686,E2 27726.686} C_VEL
LIN {X 0,Y 583.933,Z 1147.857,A -85,B 0,C 180,E1 27725.109,E2 27725.109} C_VEL
LIN {X 0,Y 583.92,Z 1153.423,A -85,B 0,C 180,E1 27723.436,E2 27723.436} C_VEL
LIN {X 0,Y 583.914,Z 1157.095,A -85,B 0,C 180,E1 27721.766,E2 27721.766} C_VEL
LIN {X 0,Y 583.914,Z 1159.066,A -85,B 0,C 180,E1 27720.098,E2 27720.098} C_VEL
LIN {X 0,Y 583.913,Z 1159.37,A -85,B 0,C 180,E1 27718.332,E2 27718.332} C_VEL
LIN {X 0,Y 583.912,Z 1157.902,A -85,B 0,C 180,E1 27716.658,E2 27716.658} C_VEL
LIN {X 0,Y 583.917,Z 1154.746,A -85,B 0,C 180,E1 27714.99,E2 27714.99} C_VEL
LIN {X 0,Y 583.93,Z 1149.404,A -85,B 0,C 180,E1 27713.215,E2 27713.215} C_VEL
LIN {X 0,Y 583.953,Z 1142.793,A -85,B 0,C 180,E1 27711.632,E2 27711.632} C_VEL
LIN {X 0,Y 583.998,Z 1134.203,A -85,B 0,C 180,E1 27710.043,E2 27710.043} C_VEL
LIN {X 0,Y 584.063,Z 1123.934,A -85,B 0,C 180,E1 27708.546,E2 27708.546} C_VEL
LIN {X 0,Y 584.143,Z 1112.964,A -85,B 0,C 180,E1 27707.244,E2 27707.244} C_VEL
LIN {X 0,Y 584.261,Z 1100.338,A -85,B 0,C 180,E1 27706.006,E2 27706.006} C_VEL
LIN {X 0,Y 584.39,Z 1086.131,A -85,B 0,C 180,E1 27704.876,E2 27704.876} C_VEL
LIN {X 0,Y 584.517,Z 1072.055,A -85,B 0,C 180,E1 27703.963,E2 27703.963} C_VEL
LIN {X 0,Y 584.643,Z 1055.169,A -85,B 0,C 180,E1 27703.098,E2 27703.098} C_VEL
LIN {X 0,Y 584.767,Z 1039.403,A -85,B 0,C 180,E1 27702.487,E2 27702.487} C_VEL
LIN {X 0,Y 584.863,Z 1022.507,A -85,B 0,C 180,E1 27702.017,E2 27702.017} C_VEL
LIN {X 0,Y 584.936,Z 1003.868,A -85,B 0,C 180,E1 27701.701,E2 27701.701} C_VEL
LIN {X 0,Y 584.963,Z 846.188,A -85,B 0,C 180,E1 27699.705,E2 27699.705} C_VEL
LIN {X 0,Y 584.775,Z 844.248,A -85,B 0,C 180,E1 27699.638,E2 27699.638} C_VEL
LIN {X 0,Y 585.105,Z 798.246,A -85,B 0,C 180,E1 27696.216,E2 27696.216} C_VEL
LIN {X 0,Y 585.465,Z 754.313,A -85,B 0,C 180,E1 27692.872,E2 27692.872} C_VEL
LIN {X 0,Y 585.862,Z 713.163,A -85,B 0,C 180,E1 27689.658,E2 27689.658} C_VEL
LIN {X 0,Y 586.31,Z 678.018,A -85,B 0,C 180,E1 27686.81,E2 27686.81} C_VEL
LIN {X 0,Y 587.747,Z 669.241,A -85,B 0,C 180,E1 27685.812,E2 27685.812} C_VEL
LIN {X 0,Y 587.159,Z 667.335,A -85,B 0,C 180,E1 27685.335,E2 27685.335} C_VEL
LIN {X 0,Y 584.764,Z 664.322,A -85,B 0,C 180,E1 27683.851,E2 27683.851} C_VEL
LIN {X 0,Y 584.217,Z 662.714,A -85,B 0,C 180,E1 27682.71,E2 27682.71} C_VEL
LIN {X 0,Y 584.281,Z 662.972,A -85,B 0,C 180,E1 27681.847,E2 27681.847} C_VEL
LIN {X 0,Y 585.086,Z 664.976,A -85,B 0,C 180,E1 27681.033,E2 27681.033} C_VEL
LIN {X 0,Y 586.598,Z 667.017,A -85,B 0,C 180,E1 27680.522,E2 27680.522} C_VEL
LIN {X 0,Y 587.234,Z 669.545,A -85,B 0,C 180,E1 27680.234,E2 27680.234} C_VEL
LIN {X 0,Y 586.04,Z 686.563,A -85,B 0,C 180,E1 27679.29,E2 27679.29} C_VEL
LIN {X 0,Y 585.353,Z 728.576,A -85,B 0,C 180,E1 27677.265,E2 27677.265} C_VEL
LIN {X 0,Y 586.474,Z 750.437,A -85,B 0,C 180,E1 27676.198,E2 27676.198} C_VEL
LIN {X 0,Y 588.554,Z 763.07,A -85,B 0,C 180,E1 27675.522,E2 27675.522} C_VEL
LIN {X 0,Y 591.232,Z 771.512,A -85,B 0,C 180,E1 27675.017,E2 27675.017} C_VEL
LIN {X 0,Y 593.686,Z 776.715,A -85,B 0,C 180,E1 27674.57,E2 27674.57} C_VEL
LIN {X 0,Y 596.429,Z 780.663,A -85,B 0,C 180,E1 27674.014,E2 27674.014} C_VEL
LIN {X 0,Y 598.449,Z 782.476,A -85,B 0,C 180,E1 27673.5,E2 27673.5} C_VEL
LIN {X 0,Y 599.9,Z 782.873,A -85,B 0,C 180,E1 27672.973,E2 27672.973} C_VEL
LIN {X 0,Y 600.636,Z 781.761,A -85,B 0,C 180,E1 27672.392,E2 27672.392} C_VEL
LIN {X 0,Y 600.325,Z 779.152,A -85,B 0,C 180,E1 27671.857,E2 27671.857} C_VEL
LIN {X 0,Y 598.972,Z 775.037,A -85,B 0,C 180,E1 27671.395,E2 27671.395} C_VEL
LIN {X 0,Y 596.842,Z 769.79,A -85,B 0,C 180,E1 27671.065,E2 27671.065} C_VEL
LIN {X 0,Y 594.304,Z 761.691,A -85,B 0,C 180,E1 27670.783,E2 27670.783} C_VEL
LIN {X 0,Y 592.675,Z 751.394,A -85,B 0,C 180,E1 27670.6,E2 27670.6} C_VEL
LIN {X 0,Y 592.05,Z 737.833,A -85,B 0,C 180,E1 27670.529,E2 27670.529} C_VEL
LIN {X 0,Y 592.024,Z 672.89,A -85,B 0,C 180,E1 27670.527,E2 27670.527} C_VEL
LIN {X 0,Y 589.11,Z 669.242,A -85,B 0,C 180,E1 27670.194,E2 27670.194} C_VEL
LIN {X 0,Y 588.305,Z 668.075,A -85,B 0,C 180,E1 27670.101,E2 27670.101} C_VEL
LIN {X 0,Y 585.576,Z 665.706,A -85,B 0,C 180,E1 27669.783,E2 27669.783} C_VEL
LIN {X 0,Y 584.488,Z 663.666,A -85,B 0,C 180,E1 27669.649,E2 27669.649} C_VEL
LIN {X 0,Y 587.954,Z 670.939,A -85,B 0,C 180,E1 27668.914,E2 27668.914} C_VEL
LIN {X 0,Y 587.368,Z 721.276,A -85,B 0,C 180,E1 27665.877,E2 27665.877} C_VEL
LIN {X 0,Y 587.097,Z 759.545,A -85,B 0,C 180,E1 27663.662,E2 27663.662} C_VEL
LIN {X 0,Y 587.702,Z 764.836,A -85,B 0,C 180,E1 27663.547,E2 27663.547} C_VEL
LIN {X 0,Y 587.023,Z 998.548,A -85,B 0,C 180,E1 27660.29,E2 27660.29} C_VEL
LIN {X 0,Y 586.803,Z 1066.129,A -85,B 0,C 180,E1 27659.336,E2 27659.336} C_VEL
LIN {X 0,Y 586.622,Z 1087.958,A -85,B 0,C 180,E1 27658.836,E2 27658.836} C_VEL
LIN {X 0,Y 586.358,Z 1110.116,A -85,B 0,C 180,E1 27658.137,E2 27658.137} C_VEL
LIN {X 0,Y 586.115,Z 1131.14,A -85,B 0,C 180,E1 27657.28,E2 27657.28} C_VEL
LIN {X 0,Y 585.823,Z 1150.743,A -85,B 0,C 180,E1 27656.29,E2 27656.29} C_VEL
LIN {X 0,Y 585.487,Z 1171.145,A -85,B 0,C 180,E1 27655.057,E2 27655.057} C_VEL
LIN {X 0,Y 585.218,Z 1189.801,A -85,B 0,C 180,E1 27653.726,E2 27653.726} C_VEL
LIN {X 0,Y 584.927,Z 1208.09,A -85,B 0,C 180,E1 27652.196,E2 27652.196} C_VEL
LIN {X 0,Y 584.667,Z 1224.19,A -85,B 0,C 180,E1 27650.628,E2 27650.628} C_VEL
LIN {X 0,Y 584.444,Z 1239.875,A -85,B 0,C 180,E1 27648.865,E2 27648.865} C_VEL
LIN {X 0,Y 584.271,Z 1254.04,A -85,B 0,C 180,E1 27647.016,E2 27647.016} C_VEL
LIN {X 0,Y 584.142,Z 1266.743,A -85,B 0,C 180,E1 27645.081,E2 27645.081} C_VEL
LIN {X 0,Y 584.045,Z 1277.852,A -85,B 0,C 180,E1 27643.061,E2 27643.061} C_VEL
LIN {X 0,Y 583.976,Z 1287.481,A -85,B 0,C 180,E1 27640.956,E2 27640.956} C_VEL
LIN {X 0,Y 583.939,Z 1295.236,A -85,B 0,C 180,E1 27638.865,E2 27638.865} C_VEL
LIN {X 0,Y 583.921,Z 1300.904,A -85,B 0,C 180,E1 27636.885,E2 27636.885} C_VEL
LIN {X 0,Y 583.908,Z 1305.47,A -85,B 0,C 180,E1 27634.715,E2 27634.715} C_VEL
LIN {X 0,Y 583.9,Z 1308.326,A -85,B 0,C 180,E1 27632.552,E2 27632.552} C_VEL
LIN {X 0,Y 583.894,Z 1309.395,A -85,B 0,C 180,E1 27630.491,E2 27630.491} C_VEL
LIN {X 0,Y 583.896,Z 1308.887,A -85,B 0,C 180,E1 27628.234,E2 27628.234} C_VEL
LIN {X 0,Y 583.896,Z 1306.866,A -85,B 0,C 180,E1 27626.171,E2 27626.171} C_VEL
LIN {X 0,Y 583.906,Z 1303.197,A -85,B 0,C 180,E1 27624.103,E2 27624.103} C_VEL
LIN {X 0,Y 583.924,Z 1297.677,A -85,B 0,C 180,E1 27621.929,E2 27621.929} C_VEL
LIN {X 0,Y 583.963,Z 1290.903,A -85,B 0,C 180,E1 27619.901,E2 27619.901} C_VEL
LIN {X 0,Y 584.011,Z 1282.224,A -85,B 0,C 180,E1 27617.844,E2 27617.844} C_VEL
LIN {X 0,Y 584.097,Z 1271.97,A -85,B 0,C 180,E1 27615.831,E2 27615.831} C_VEL
LIN {X 0,Y 584.192,Z 1260.98,A -85,B 0,C 180,E1 27614.005,E2 27614.005} C_VEL
LIN {X 0,Y 584.336,Z 1248.024,A -85,B 0,C 180,E1 27612.165,E2 27612.165} C_VEL
LIN {X 0,Y 584.535,Z 1233.738,A -85,B 0,C 180,E1 27610.412,E2 27610.412} C_VEL
LIN {X 0,Y 584.781,Z 1217.849,A -85,B 0,C 180,E1 27608.723,E2 27608.723} C_VEL
LIN {X 0,Y 585.06,Z 1199.656,A -85,B 0,C 180,E1 27607.068,E2 27607.068} C_VEL
LIN {X 0,Y 585.333,Z 1181.214,A -85,B 0,C 180,E1 27605.637,E2 27605.637} C_VEL
LIN {X 0,Y 585.65,Z 1161.735,A -85,B 0,C 180,E1 27604.347,E2 27604.347} C_VEL
LIN {X 0,Y 585.967,Z 1141.646,A -85,B 0,C 180,E1 27603.227,E2 27603.227} C_VEL
LIN {X 0,Y 586.229,Z 1121.414,A -85,B 0,C 180,E1 27602.3,E2 27602.3} C_VEL
LIN {X 0,Y 586.487,Z 1100.078,A -85,B 0,C 180,E1 27601.523,E2 27601.523} C_VEL
LIN {X 0,Y 586.717,Z 1078.342,A -85,B 0,C 180,E1 27600.919,E2 27600.919} C_VEL
LIN {X 0,Y 586.84,Z 1056.46,A -85,B 0,C 180,E1 27600.506,E2 27600.506} C_VEL
LIN {X 0,Y 587.503,Z 827.673,A -85,B 0,C 180,E1 27597.339,E2 27597.339} C_VEL
LIN {X 0,Y 587.507,Z 761.925,A -85,B 0,C 180,E1 27596.399,E2 27596.399} C_VEL
LIN {X 0,Y 586.983,Z 758.576,A -85,B 0,C 180,E1 27596.306,E2 27596.306} C_VEL
LIN {X 0,Y 587.553,Z 705.798,A -85,B 0,C 180,E1 27593.202,E2 27593.202} C_VEL
LIN {X 0,Y 587.954,Z 670.94,A -85,B 0,C 180,E1 27591.086,E2 27591.086} C_VEL
LIN {X 0,Y 584.493,Z 663.675,A -85,B 0,C 180,E1 27590.345,E2 27590.345} C_VEL
LIN {X 0,Y 586.372,Z 666.643,A -85,B 0,C 180,E1 27590.124,E2 27590.124} C_VEL
LIN {X 0,Y 588.782,Z 668.634,A -85,B 0,C 180,E1 27589.844,E2 27589.844} C_VEL
LIN {X 0,Y 591.532,Z 672.427,A -85,B 0,C 180,E1 27589.529,E2 27589.529} C_VEL
LIN {X 0,Y 592.042,Z 672.905,A -85,B 0,C 180,E1 27589.472,E2 27589.472} C_VEL
LIN {X 0,Y 592.227,Z 745.048,A -85,B 0,C 180,E1 27589.451,E2 27589.451} C_VEL
LIN {X 0,Y 593.341,Z 756.657,A -85,B 0,C 180,E1 27589.325,E2 27589.325} C_VEL
LIN {X 0,Y 595.361,Z 765.612,A -85,B 0,C 180,E1 27589.099,E2 27589.099} C_VEL
LIN {X 0,Y 598.025,Z 772.641,A -85,B 0,C 180,E1 27588.781,E2 27588.781} C_VEL
LIN {X 0,Y 599.777,Z 777.238,A -85,B 0,C 180,E1 27588.387,E2 27588.387} C_VEL
LIN {X 0,Y 600.6,Z 780.511,A -85,B 0,C 180,E1 27587.907,E2 27587.907} C_VEL
LIN {X 0,Y 600.475,Z 782.374,A -85,B 0,C 180,E1 27587.39,E2 27587.39} C_VEL
LIN {X 0,Y 599.36,Z 782.884,A -85,B 0,C 180,E1 27586.803,E2 27586.803} C_VEL
LIN {X 0,Y 597.654,Z 781.874,A -85,B 0,C 180,E1 27586.279,E2 27586.279} C_VEL
LIN {X 0,Y 595.554,Z 779.577,A -85,B 0,C 180,E1 27585.797,E2 27585.797} C_VEL
LIN {X 0,Y 592.775,Z 774.929,A -85,B 0,C 180,E1 27585.244,E2 27585.244} C_VEL
LIN {X 0,Y 590.205,Z 766.671,A -85,B 0,C 180,E1 27584.504,E2 27584.504} C_VEL
LIN {X 0,Y 588.881,Z 755.547,A -85,B 0,C 180,E1 27583.673,E2 27583.673} C_VEL
LIN {X 0,Y 589.336,Z 701.463,A -85,B 0,C 180,E1 27580.08,E2 27580.08} C_VEL
LIN {X 0,Y 589.693,Z 673.441,A -85,B 0,C 180,E1 27578.11,E2 27578.11} C_VEL
LIN {X 0,Y 588.197,Z 670.496,A -85,B 0,C 180,E1 27577.731,E2 27577.731} C_VEL
LIN {X 0,Y 585.953,Z 666.184,A -85,B 0,C 180,E1 27577.161,E2 27577.161} C_VEL
LIN {X 0,Y 584.29,Z 662.983,A -85,B 0,C 180,E1 27576.732,E2 27576.732} C_VEL
LIN {X 0,Y 584.097,Z 661.982,A -85,B 0,C 180,E1 27576.599,E2 27576.599} C_VEL
LIN {X 0,Y 584.095,Z 661.982,A -85,B 0,C 180,E1 27573.332,E2 27573.332} C_VEL
LIN {X 0,Y 584.079,Z 661.981,A -85,B 0,C 180,E1 27570.104,E2 27570.104} C_VEL
LIN {X 0,Y 584.084,Z 661.978,A -85,B 0,C 180,E1 27566.977,E2 27566.977} C_VEL
LIN {X 0,Y 584.079,Z 661.978,A -85,B 0,C 180,E1 27563.828,E2 27563.828} C_VEL
LIN {X 0,Y 584.08,Z 661.978,A -85,B 0,C 180,E1 27560.649,E2 27560.649} C_VEL
LIN {X 0,Y 584.08,Z 661.978,A -85,B 0,C 180,E1 27557.432,E2 27557.432} C_VEL
LIN {X 0,Y 584.085,Z 661.978,A -85,B 0,C 180,E1 27554.271,E2 27554.271} C_VEL
LIN {X 0,Y 584.088,Z 661.977,A -85,B 0,C 180,E1 27551.053,E2 27551.053} C_VEL
LIN {X 0,Y 584.083,Z 661.978,A -85,B 0,C 180,E1 27547.772,E2 27547.772} C_VEL
LIN {X 0,Y 584.095,Z 661.979,A -85,B 0,C 180,E1 27544.516,E2 27544.516} C_VEL
LIN {X 0,Y 584.097,Z 661.982,A -85,B 0,C 180,E1 27541.177,E2 27541.177} C_VEL
LIN {X 0,Y 584.087,Z 661.982,A -85,B 0,C 180,E1 27537.94,E2 27537.94} C_VEL
LIN {X 0,Y 584.088,Z 661.979,A -85,B 0,C 180,E1 27534.696,E2 27534.696} C_VEL
LIN {X 0,Y 584.078,Z 661.979,A -85,B 0,C 180,E1 27531.435,E2 27531.435} C_VEL
LIN {X 0,Y 584.078,Z 661.979,A -85,B 0,C 180,E1 27528.246,E2 27528.246} C_VEL
LIN {X 0,Y 584.088,Z 661.977,A -85,B 0,C 180,E1 27526.719,E2 27526.719} C_VEL
LIN {X 0,Y 583.118,Z 662.101,A -85,B 0,C 180,E1 27525.964,E2 27525.964} C_VEL
LIN {X 0,Y 576.685,Z 662.902,A -85,B 0,C 180,E1 27523.843,E2 27523.843} C_VEL
LIN {X 0,Y 576.159,Z 662.965,A -85,B 0,C 180,E1 27523.291,E2 27523.291} C_VEL
LIN {X 0,Y 576.151,Z 662.966,A -85,B 0,C 180,E1 27519.858,E2 27519.858} C_VEL
LIN {X 0,Y 576.161,Z 662.967,A -85,B 0,C 180,E1 27516.584,E2 27516.584} C_VEL
LIN {X 0,Y 576.156,Z 662.966,A -85,B 0,C 180,E1 27513.29,E2 27513.29} C_VEL
LIN {X 0,Y 576.143,Z 662.966,A -85,B 0,C 180,E1 27509.994,E2 27509.994} C_VEL
LIN {X 0,Y 576.141,Z 662.967,A -85,B 0,C 180,E1 27506.743,E2 27506.743} C_VEL
LIN {X 0,Y 576.144,Z 662.965,A -85,B 0,C 180,E1 27503.593,E2 27503.593} C_VEL
LIN {X 0,Y 576.146,Z 662.964,A -85,B 0,C 180,E1 27500.4,E2 27500.4} C_VEL
LIN {X 0,Y 576.143,Z 662.967,A -85,B 0,C 180,E1 27497.083,E2 27497.083} C_VEL
LIN {X 0,Y 576.141,Z 662.97,A -85,B 0,C 180,E1 27493.823,E2 27493.823} C_VEL
LIN {X 0,Y 576.155,Z 662.972,A -85,B 0,C 180,E1 27490.526,E2 27490.526} C_VEL
LIN {X 0,Y 576.158,Z 662.969,A -85,B 0,C 180,E1 27487.198,E2 27487.198} C_VEL
LIN {X 0,Y 576.143,Z 662.979,A -85,B 0,C 180,E1 27486.198,E2 27486.198} C_VEL
LIN {X 0,Y 580.079,Z 673.205,A -85,B 0,C 180,E1 27485.213,E2 27485.213} C_VEL
LIN {X 0,Y 579.423,Z 719.052,A -85,B 0,C 180,E1 27482.164,E2 27482.164} C_VEL
LIN {X 0,Y 578.906,Z 765.983,A -85,B 0,C 180,E1 27479.154,E2 27479.154} C_VEL
LIN {X 0,Y 579.669,Z 772.295,A -85,B 0,C 180,E1 27479.024,E2 27479.024} C_VEL
LIN {X 0,Y 578.91,Z 1008.772,A -85,B 0,C 180,E1 27475.826,E2 27475.826} C_VEL
LIN {X 0,Y 578.775,Z 1033.57,A -85,B 0,C 180,E1 27475.432,E2 27475.432} C_VEL
LIN {X 0,Y 578.554,Z 1054.048,A -85,B 0,C 180,E1 27474.918,E2 27474.918} C_VEL
LIN {X 0,Y 578.299,Z 1074.285,A -85,B 0,C 180,E1 27474.217,E2 27474.217} C_VEL
LIN {X 0,Y 577.989,Z 1093.87,A -85,B 0,C 180,E1 27473.337,E2 27473.337} C_VEL
LIN {X 0,Y 577.665,Z 1112.055,A -85,B 0,C 180,E1 27472.328,E2 27472.328} C_VEL
LIN {X 0,Y 577.321,Z 1130.257,A -85,B 0,C 180,E1 27471.114,E2 27471.114} C_VEL
LIN {X 0,Y 576.993,Z 1148.025,A -85,B 0,C 180,E1 27469.696,E2 27469.696} C_VEL
LIN {X 0,Y 576.707,Z 1164.485,A -85,B 0,C 180,E1 27468.137,E2 27468.137} C_VEL
LIN {X 0,Y 576.468,Z 1178.896,A -85,B 0,C 180,E1 27466.525,E2 27466.525} C_VEL
LIN {X 0,Y 576.273,Z 1192.18,A -85,B 0,C 180,E1 27464.776,E2 27464.776} C_VEL
LIN {X 0,Y 576.143,Z 1203.36,A -85,B 0,C 180,E1 27463.038,E2 27463.038} C_VEL
LIN {X 0,Y 576.041,Z 1213.693,A -85,B 0,C 180,E1 27461.108,E2 27461.108} C_VEL
LIN {X 0,Y 575.963,Z 1222.011,A -85,B 0,C 180,E1 27459.19,E2 27459.19} C_VEL
LIN {X 0,Y 575.924,Z 1228.571,A -85,B 0,C 180,E1 27457.28,E2 27457.28} C_VEL
LIN {X 0,Y 575.914,Z 1233.757,A -85,B 0,C 180,E1 27455.279,E2 27455.279} C_VEL
LIN {X 0,Y 575.914,Z 1237.28,A -85,B 0,C 180,E1 27453.284,E2 27453.284} C_VEL
LIN {X 0,Y 575.904,Z 1239.109,A -85,B 0,C 180,E1 27451.293,E2 27451.293} C_VEL
LIN {X 0,Y 575.903,Z 1239.361,A -85,B 0,C 180,E1 27449.303,E2 27449.303} C_VEL
LIN {X 0,Y 575.912,Z 1237.942,A -85,B 0,C 180,E1 27447.213,E2 27447.213} C_VEL
LIN {X 0,Y 575.921,Z 1234.964,A -85,B 0,C 180,E1 27445.219,E2 27445.219} C_VEL
LIN {X 0,Y 575.932,Z 1230.334,A -85,B 0,C 180,E1 27443.22,E2 27443.22} C_VEL
LIN {X 0,Y 575.956,Z 1223.864,A -85,B 0,C 180,E1 27441.212,E2 27441.212} C_VEL
LIN {X 0,Y 576.014,Z 1215.794,A -85,B 0,C 180,E1 27439.259,E2 27439.259} C_VEL
LIN {X 0,Y 576.095,Z 1206.174,A -85,B 0,C 180,E1 27437.368,E2 27437.368} C_VEL
LIN {X 0,Y 576.24,Z 1194.802,A -85,B 0,C 180,E1 27435.515,E2 27435.515} C_VEL
LIN {X 0,Y 576.425,Z 1182.151,A -85,B 0,C 180,E1 27433.783,E2 27433.783} C_VEL
LIN {X 0,Y 576.659,Z 1167.902,A -85,B 0,C 180,E1 27432.127,E2 27432.127} C_VEL
LIN {X 0,Y 576.945,Z 1152.039,A -85,B 0,C 180,E1 27430.564,E2 27430.564} C_VEL
LIN {X 0,Y 577.252,Z 1135.318,A -85,B 0,C 180,E1 27429.171,E2 27429.171} C_VEL
LIN {X 0,Y 577.567,Z 1117.71,A -85,B 0,C 180,E1 27427.935,E2 27427.935} C_VEL
LIN {X 0,Y 577.864,Z 1099.62,A -85,B 0,C 180,E1 27426.873,E2 27426.873} C_VEL
LIN {X 0,Y 578.196,Z 1079.561,A -85,B 0,C 180,E1 27425.914,E2 27425.914} C_VEL
LIN {X 0,Y 578.509,Z 1059.05,A -85,B 0,C 180,E1 27425.149,E2 27425.149} C_VEL
LIN {X 0,Y 578.735,Z 1038.556,A -85,B 0,C 180,E1 27424.585,E2 27424.585} C_VEL
LIN {X 0,Y 578.881,Z 1017.667,A -85,B 0,C 180,E1 27424.203,E2 27424.203} C_VEL
LIN {X 0,Y 579.636,Z 782.352,A -85,B 0,C 180,E1 27421.023,E2 27421.023} C_VEL
LIN {X 0,Y 579.446,Z 772.767,A -85,B 0,C 180,E1 27420.88,E2 27420.88} C_VEL
LIN {X 0,Y 578.231,Z 767.505,A -85,B 0,C 180,E1 27420.73,E2 27420.73} C_VEL
LIN {X 0,Y 578.739,Z 733.058,A -85,B 0,C 180,E1 27417.558,E2 27417.558} C_VEL
LIN {X 0,Y 579.299,Z 699.664,A -85,B 0,C 180,E1 27414.384,E2 27414.384} C_VEL
LIN {X 0,Y 579.531,Z 672.913,A -85,B 0,C 180,E1 27411.809,E2 27411.809} C_VEL
LIN {X 0,Y 576.14,Z 662.971,A -85,B 0,C 180,E1 27410.599,E2 27410.599} C_VEL
LIN {X 0,Y 576.14,Z 662.968,A -85,B 0,C 180,E1 27407.377,E2 27407.377} C_VEL
LIN {X 0,Y 576.156,Z 662.97,A -85,B 0,C 180,E1 27404.099,E2 27404.099} C_VEL
LIN {X 0,Y 576.141,Z 662.962,A -85,B 0,C 180,E1 27400.83,E2 27400.83} C_VEL
LIN {X 0,Y 576.142,Z 662.972,A -85,B 0,C 180,E1 27397.653,E2 27397.653} C_VEL
LIN {X 0,Y 576.139,Z 662.969,A -85,B 0,C 180,E1 27394.455,E2 27394.455} C_VEL
LIN {X 0,Y 576.162,Z 663.059,A -85,B 0,C 180,E1 27393.051,E2 27393.051} C_VEL
LIN {X 0,Y 579.223,Z 672.48,A -85,B 0,C 180,E1 27392.002,E2 27392.002} C_VEL
LIN {X 0,Y 578.604,Z 709.001,A -85,B 0,C 180,E1 27388.994,E2 27388.994} C_VEL
LIN {X 0,Y 578.067,Z 749.386,A -85,B 0,C 180,E1 27385.786,E2 27385.786} C_VEL
LIN {X 0,Y 577.6,Z 790.516,A -85,B 0,C 180,E1 27382.6,E2 27382.6} C_VEL
LIN {X 0,Y 577.178,Z 833.788,A -85,B 0,C 180,E1 27379.322,E2 27379.322} C_VEL
LIN {X 0,Y 577.131,Z 845.208,A -85,B 0,C 180,E1 27378.489,E2 27378.489} C_VEL
LIN {X 0,Y 577.6,Z 851.709,A -85,B 0,C 180,E1 27378.389,E2 27378.389} C_VEL
LIN {X 0,Y 577.236,Z 1015.209,A -85,B 0,C 180,E1 27376.274,E2 27376.274} C_VEL
LIN {X 0,Y 577.129,Z 1033.553,A -85,B 0,C 180,E1 27375.835,E2 27375.835} C_VEL
LIN {X 0,Y 576.979,Z 1049.458,A -85,B 0,C 180,E1 27375.272,E2 27375.272} C_VEL
LIN {X 0,Y 576.808,Z 1064.8,A -85,B 0,C 180,E1 27374.557,E2 27374.557} C_VEL
LIN {X 0,Y 576.633,Z 1080.288,A -85,B 0,C 180,E1 27373.64,E2 27373.64} C_VEL
LIN {X 0,Y 576.453,Z 1094.61,A -85,B 0,C 180,E1 27372.573,E2 27372.573} C_VEL
LIN {X 0,Y 576.295,Z 1107.524,A -85,B 0,C 180,E1 27371.402,E2 27371.402} C_VEL
LIN {X 0,Y 576.154,Z 1120.175,A -85,B 0,C 180,E1 27369.994,E2 27369.994} C_VEL
LIN {X 0,Y 576.057,Z 1130.448,A -85,B 0,C 180,E1 27368.585,E2 27368.585} C_VEL
LIN {X 0,Y 575.983,Z 1139.838,A -85,B 0,C 180,E1 27366.98,E2 27366.98} C_VEL
LIN {X 0,Y 575.941,Z 1147.125,A -85,B 0,C 180,E1 27365.379,E2 27365.379} C_VEL
LIN {X 0,Y 575.925,Z 1152.589,A -85,B 0,C 180,E1 27363.783,E2 27363.783} C_VEL
LIN {X 0,Y 575.916,Z 1156.633,A -85,B 0,C 180,E1 27362.09,E2 27362.09} C_VEL
LIN {X 0,Y 575.914,Z 1158.861,A -85,B 0,C 180,E1 27360.398,E2 27360.398} C_VEL
LIN {X 0,Y 575.912,Z 1159.457,A -85,B 0,C 180,E1 27358.707,E2 27358.707} C_VEL
LIN {X 0,Y 575.911,Z 1158.156,A -85,B 0,C 180,E1 27356.815,E2 27356.815} C_VEL
LIN {X 0,Y 575.919,Z 1155.165,A -85,B 0,C 180,E1 27355.12,E2 27355.12} C_VEL
LIN {X 0,Y 575.931,Z 1150.413,A -85,B 0,C 180,E1 27353.421,E2 27353.421} C_VEL
LIN {X 0,Y 575.96,Z 1143.556,A -85,B 0,C 180,E1 27351.696,E2 27351.696} C_VEL
LIN {X 0,Y 576.006,Z 1135.846,A -85,B 0,C 180,E1 27350.206,E2 27350.206} C_VEL
LIN {X 0,Y 576.097,Z 1126.09,A -85,B 0,C 180,E1 27348.69,E2 27348.69} C_VEL
LIN {X 0,Y 576.212,Z 1114.671,A -85,B 0,C 180,E1 27347.269,E2 27347.269} C_VEL
LIN {X 0,Y 576.355,Z 1102.425,A -85,B 0,C 180,E1 27346.018,E2 27346.018} C_VEL
LIN {X 0,Y 576.549,Z 1087.589,A -85,B 0,C 180,E1 27344.784,E2 27344.784} C_VEL
LIN {X 0,Y 576.714,Z 1073.417,A -85,B 0,C 180,E1 27343.839,E2 27343.839} C_VEL
LIN {X 0,Y 576.891,Z 1058.221,A -85,B 0,C 180,E1 27343.02,E2 27343.02} C_VEL
LIN {X 0,Y 577.062,Z 1040.459,A -85,B 0,C 180,E1 27342.297,E2 27342.297} C_VEL
LIN {X 0,Y 577.184,Z 1023.846,A -85,B 0,C 180,E1 27341.819,E2 27341.819} C_VEL
LIN {X 0,Y 577.292,Z 1006.202,A -85,B 0,C 180,E1 27341.495,E2 27341.495} C_VEL
LIN {X 0,Y 577.401,Z 847.088,A -85,B 0,C 180,E1 27339.455,E2 27339.455} C_VEL
LIN {X 0,Y 577.083,Z 844.745,A -85,B 0,C 180,E1 27339.408,E2 27339.408} C_VEL
LIN {X 0,Y 577.518,Z 799.45,A -85,B 0,C 180,E1 27335.993,E2 27335.993} C_VEL
LIN {X 0,Y 578.006,Z 755.517,A -85,B 0,C 180,E1 27332.604,E2 27332.604} C_VEL
LIN {X 0,Y 578.538,Z 714.366,A -85,B 0,C 180,E1 27329.347,E2 27329.347} C_VEL
LIN {X 0,Y 578.854,Z 696.971,A -85,B 0,C 180,E1 27327.917,E2 27327.917} C_VEL
LIN {X 0,Y 582.038,Z 678.128,A -85,B 0,C 180,E1 27325.895,E2 27325.895} C_VEL
LIN {X 0,Y 582.766,Z 674.847,A -85,B 0,C 180,E1 27325.516,E2 27325.516} C_VEL
LIN {X 0,Y 582.194,Z 673.557,A -85,B 0,C 180,E1 27325.118,E2 27325.118} C_VEL
LIN {X 0,Y 580.122,Z 670.576,A -85,B 0,C 180,E1 27323.6,E2 27323.6} C_VEL
LIN {X 0,Y 579.823,Z 669.342,A -85,B 0,C 180,E1 27322.489,E2 27322.489} C_VEL
LIN {X 0,Y 580.018,Z 670.107,A -85,B 0,C 180,E1 27321.642,E2 27321.642} C_VEL
LIN {X 0,Y 581.133,Z 672.43,A -85,B 0,C 180,E1 27320.844,E2 27320.844} C_VEL
LIN {X 0,Y 581.474,Z 673.575,A -85,B 0,C 180,E1 27320.645,E2 27320.645} C_VEL
LIN {X 0,Y 579.63,Z 686.203,A -85,B 0,C 180,E1 27319.824,E2 27319.824} C_VEL
LIN {X 0,Y 578.383,Z 707.326,A -85,B 0,C 180,E1 27318.672,E2 27318.672} C_VEL
LIN {X 0,Y 578.199,Z 740.579,A -85,B 0,C 180,E1 27317.011,E2 27317.011} C_VEL
LIN {X 0,Y 579.733,Z 758.093,A -85,B 0,C 180,E1 27316.106,E2 27316.106} C_VEL
LIN {X 0,Y 582.503,Z 770.505,A -85,B 0,C 180,E1 27315.409,E2 27315.409} C_VEL
LIN {X 0,Y 586.378,Z 779.753,A -85,B 0,C 180,E1 27314.819,E2 27314.819} C_VEL
LIN {X 0,Y 589.381,Z 784.399,A -85,B 0,C 180,E1 27314.422,E2 27314.422} C_VEL
LIN {X 0,Y 592.778,Z 788.106,A -85,B 0,C 180,E1 27313.888,E2 27313.888} C_VEL
LIN {X 0,Y 595.384,Z 789.897,A -85,B 0,C 180,E1 27313.352,E2 27313.352} C_VEL
LIN {X 0,Y 597.153,Z 790.249,A -85,B 0,C 180,E1 27312.828,E2 27312.828} C_VEL
LIN {X 0,Y 598.182,Z 789.205,A -85,B 0,C 180,E1 27312.229,E2 27312.229} C_VEL
LIN {X 0,Y 598.008,Z 786.706,A -85,B 0,C 180,E1 27311.653,E2 27311.653} C_VEL
LIN {X 0,Y 596.704,Z 783.026,A -85,B 0,C 180,E1 27311.172,E2 27311.172} C_VEL
LIN {X 0,Y 594.384,Z 778.273,A -85,B 0,C 180,E1 27310.792,E2 27310.792} C_VEL
LIN {X 0,Y 591.091,Z 770.452,A -85,B 0,C 180,E1 27310.421,E2 27310.421} C_VEL
LIN {X 0,Y 588.728,Z 761.049,A -85,B 0,C 180,E1 27310.15,E2 27310.15} C_VEL
LIN {X 0,Y 587.3,Z 749.534,A -85,B 0,C 180,E1 27309.984,E2 27309.984} C_VEL
LIN {X 0,Y 586.884,Z 737.989,A -85,B 0,C 180,E1 27309.936,E2 27309.936} C_VEL
LIN {X 0,Y 586.778,Z 676.888,A -85,B 0,C 180,E1 27309.924,E2 27309.924} C_VEL
LIN {X 0,Y 584.937,Z 674.548,A -85,B 0,C 180,E1 27309.708,E2 27309.708} C_VEL
LIN {X 0,Y 584.458,Z 674.308,A -85,B 0,C 180,E1 27309.651,E2 27309.651} C_VEL
LIN {X 0,Y 582.549,Z 674.785,A -85,B 0,C 180,E1 27309.424,E2 27309.424} C_VEL
LIN {X 0,Y 581.218,Z 674.344,A -85,B 0,C 180,E1 27309.235,E2 27309.235} C_VEL
LIN {X 0,Y 580.701,Z 714.805,A -85,B 0,C 180,E1 27306.751,E2 27306.751} C_VEL
LIN {X 0,Y 580.193,Z 759.527,A -85,B 0,C 180,E1 27304.117,E2 27304.117} C_VEL
LIN {X 0,Y 581.026,Z 766.086,A -85,B 0,C 180,E1 27303.966,E2 27303.966} C_VEL
LIN {X 0,Y 580.108,Z 1000.007,A -85,B 0,C 180,E1 27300.669,E2 27300.669} C_VEL
LIN {X 0,Y 579.821,Z 1066.116,A -85,B 0,C 180,E1 27299.725,E2 27299.725} C_VEL
LIN {X 0,Y 579.574,Z 1088.201,A -85,B 0,C 180,E1 27299.214,E2 27299.214} C_VEL
LIN {X 0,Y 579.22,Z 1110.803,A -85,B 0,C 180,E1 27298.489,E2 27298.489} C_VEL
LIN {X 0,Y 578.888,Z 1131.802,A -85,B 0,C 180,E1 27297.619,E2 27297.619} C_VEL
LIN {X 0,Y 578.489,Z 1151.744,A -85,B 0,C 180,E1 27296.594,E2 27296.594} C_VEL
LIN {X 0,Y 578.067,Z 1171.15,A -85,B 0,C 180,E1 27295.402,E2 27295.402} C_VEL
LIN {X 0,Y 577.691,Z 1189.798,A -85,B 0,C 180,E1 27294.054,E2 27294.054} C_VEL
LIN {X 0,Y 577.288,Z 1208.081,A -85,B 0,C 180,E1 27292.506,E2 27292.506} C_VEL
LIN {X 0,Y 576.942,Z 1224.189,A -85,B 0,C 180,E1 27290.917,E2 27290.917} C_VEL
LIN {X 0,Y 576.639,Z 1240.189,A -85,B 0,C 180,E1 27289.092,E2 27289.092} C_VEL
LIN {X 0,Y 576.411,Z 1254.043,A -85,B 0,C 180,E1 27287.255,E2 27287.255} C_VEL
LIN {X 0,Y 576.231,Z 1266.948,A -85,B 0,C 180,E1 27285.258,E2 27285.258} C_VEL
LIN {X 0,Y 576.095,Z 1277.854,A -85,B 0,C 180,E1 27283.244,E2 27283.244} C_VEL
LIN {X 0,Y 576.002,Z 1287.484,A -85,B 0,C 180,E1 27281.11,E2 27281.11} C_VEL
LIN {X 0,Y 575.953,Z 1295.307,A -85,B 0,C 180,E1 27278.965,E2 27278.965} C_VEL
LIN {X 0,Y 575.923,Z 1300.904,A -85,B 0,C 180,E1 27276.981,E2 27276.981} C_VEL
LIN {X 0,Y 575.907,Z 1305.497,A -85,B 0,C 180,E1 27274.766,E2 27274.766} C_VEL
LIN {X 0,Y 575.899,Z 1308.322,A -85,B 0,C 180,E1 27272.588,E2 27272.588} C_VEL
LIN {X 0,Y 575.894,Z 1309.395,A -85,B 0,C 180,E1 27270.498,E2 27270.498} C_VEL
LIN {X 0,Y 575.897,Z 1308.889,A -85,B 0,C 180,E1 27268.21,E2 27268.21} C_VEL
LIN {X 0,Y 575.897,Z 1306.862,A -85,B 0,C 180,E1 27266.118,E2 27266.118} C_VEL
LIN {X 0,Y 575.904,Z 1303.198,A -85,B 0,C 180,E1 27264.021,E2 27264.021} C_VEL
LIN {X 0,Y 575.926,Z 1297.678,A -85,B 0,C 180,E1 27261.816,E2 27261.816} C_VEL
LIN {X 0,Y 575.975,Z 1291.052,A -85,B 0,C 180,E1 27259.802,E2 27259.802} C_VEL
LIN {X 0,Y 576.043,Z 1282.557,A -85,B 0,C 180,E1 27257.746,E2 27257.746} C_VEL
LIN {X 0,Y 576.158,Z 1272.545,A -85,B 0,C 180,E1 27255.734,E2 27255.734} C_VEL
LIN {X 0,Y 576.292,Z 1261.624,A -85,B 0,C 180,E1 27253.884,E2 27253.884} C_VEL
LIN {X 0,Y 576.503,Z 1248.028,A -85,B 0,C 180,E1 27251.914,E2 27251.914} C_VEL
LIN {X 0,Y 576.76,Z 1233.735,A -85,B 0,C 180,E1 27250.137,E2 27250.137} C_VEL
LIN {X 0,Y 577.084,Z 1218.092,A -85,B 0,C 180,E1 27248.451,E2 27248.451} C_VEL
LIN {X 0,Y 577.478,Z 1199.653,A -85,B 0,C 180,E1 27246.749,E2 27246.749} C_VEL
LIN {X 0,Y 577.839,Z 1181.944,A -85,B 0,C 180,E1 27245.355,E2 27245.355} C_VEL
LIN {X 0,Y 578.265,Z 1161.891,A -85,B 0,C 180,E1 27244.004,E2 27244.004} C_VEL
LIN {X 0,Y 578.694,Z 1141.646,A -85,B 0,C 180,E1 27242.863,E2 27242.863} C_VEL
LIN {X 0,Y 579.066,Z 1121.362,A -85,B 0,C 180,E1 27241.924,E2 27241.924} C_VEL
LIN {X 0,Y 579.398,Z 1099.976,A -85,B 0,C 180,E1 27241.138,E2 27241.138} C_VEL
LIN {X 0,Y 579.71,Z 1077.891,A -85,B 0,C 180,E1 27240.522,E2 27240.522} C_VEL
LIN {X 0,Y 579.876,Z 1055.875,A -85,B 0,C 180,E1 27240.107,E2 27240.107} C_VEL
LIN {X 0,Y 580.762,Z 828.436,A -85,B 0,C 180,E1 27236.922,E2 27236.922} C_VEL
LIN {X 0,Y 580.833,Z 763.301,A -85,B 0,C 180,E1 27235.98,E2 27235.98} C_VEL
LIN {X 0,Y 580.094,Z 758.142,A -85,B 0,C 180,E1 27235.826,E2 27235.826} C_VEL
LIN {X 0,Y 580.858,Z 704.896,A -85,B 0,C 180,E1 27232.65,E2 27232.65} C_VEL
LIN {X 0,Y 581.219,Z 674.342,A -85,B 0,C 180,E1 27230.764,E2 27230.764} C_VEL
LIN {X 0,Y 583.179,Z 674.776,A -85,B 0,C 180,E1 27230.501,E2 27230.501} C_VEL
LIN {X 0,Y 584.772,Z 674.418,A -85,B 0,C 180,E1 27230.312,E2 27230.312} C_VEL
LIN {X 0,Y 586.211,Z 676.085,A -85,B 0,C 180,E1 27230.143,E2 27230.143} C_VEL
LIN {X 0,Y 586.876,Z 677.018,A -85,B 0,C 180,E1 27230.065,E2 27230.065} C_VEL
LIN {X 0,Y 587.064,Z 745.46,A -85,B 0,C 180,E1 27230.043,E2 27230.043} C_VEL
LIN {X 0,Y 588.199,Z 757.858,A -85,B 0,C 180,E1 27229.911,E2 27229.911} C_VEL
LIN {X 0,Y 590.276,Z 767.77,A -85,B 0,C 180,E1 27229.672,E2 27229.672} C_VEL
LIN {X 0,Y 593.32,Z 776.106,A -85,B 0,C 180,E1 27229.327,E2 27229.327} C_VEL
LIN {X 0,Y 596.104,Z 781.729,A -85,B 0,C 180,E1 27228.954,E2 27228.954} C_VEL
LIN {X 0,Y 597.759,Z 785.818,A -85,B 0,C 180,E1 27228.487,E2 27228.487} C_VEL
LIN {X 0,Y 598.259,Z 788.6,A -85,B 0,C 180,E1 27227.952,E2 27227.952} C_VEL
LIN {X 0,Y 597.668,Z 790.046,A -85,B 0,C 180,E1 27227.399,E2 27227.399} C_VEL
LIN {X 0,Y 595.997,Z 790.146,A -85,B 0,C 180,E1 27226.807,E2 27226.807} C_VEL
LIN {X 0,Y 593.619,Z 788.795,A -85,B 0,C 180,E1 27226.268,E2 27226.268} C_VEL
LIN {X 0,Y 590.514,Z 785.806,A -85,B 0,C 180,E1 27225.743,E2 27225.743} C_VEL
LIN {X 0,Y 586.778,Z 779.922,A -85,B 0,C 180,E1 27225.072,E2 27225.072} C_VEL
LIN {X 0,Y 584.076,Z 771.581,A -85,B 0,C 180,E1 27224.302,E2 27224.302} C_VEL
LIN {X 0,Y 582.576,Z 760.199,A -85,B 0,C 180,E1 27223.422,E2 27223.422} C_VEL
LIN {X 0,Y 582.522,Z 738.389,A -85,B 0,C 180,E1 27221.962,E2 27221.962} C_VEL
LIN {X 0,Y 583.241,Z 701.94,A -85,B 0,C 180,E1 27219.495,E2 27219.495} C_VEL
LIN {X 0,Y 583.652,Z 677.661,A -85,B 0,C 180,E1 27217.766,E2 27217.766} C_VEL
LIN {X 0,Y 580.028,Z 671.084,A -85,B 0,C 180,E1 27216.861,E2 27216.861} C_VEL
LIN {X 0,Y 578.247,Z 667.45,A -85,B 0,C 180,E1 27216.376,E2 27216.376} C_VEL
LIN {X 0,Y 576.368,Z 664.077,A -85,B 0,C 180,E1 27215.892,E2 27215.892} C_VEL
LIN {X 0,Y 576.144,Z 662.971,A -85,B 0,C 180,E1 27215.761,E2 27215.761} C_VEL
LIN {X 0,Y 576.149,Z 662.969,A -85,B 0,C 180,E1 27212.499,E2 27212.499} C_VEL
LIN {X 0,Y 576.144,Z 662.97,A -85,B 0,C 180,E1 27209.3,E2 27209.3} C_VEL
LIN {X 0,Y 576.16,Z 662.967,A -85,B 0,C 180,E1 27205.984,E2 27205.984} C_VEL
LIN {X 0,Y 576.158,Z 662.968,A -85,B 0,C 180,E1 27202.599,E2 27202.599} C_VEL
LIN {X 0,Y 576.141,Z 662.969,A -85,B 0,C 180,E1 27199.358,E2 27199.358} C_VEL
LIN {X 0,Y 576.145,Z 662.968,A -85,B 0,C 180,E1 27196.121,E2 27196.121} C_VEL
LIN {X 0,Y 576.14,Z 662.968,A -85,B 0,C 180,E1 27192.834,E2 27192.834} C_VEL
LIN {X 0,Y 576.139,Z 662.967,A -85,B 0,C 180,E1 27189.691,E2 27189.691} C_VEL
LIN {X 0,Y 576.139,Z 662.966,A -85,B 0,C 180,E1 27186.477,E2 27186.477} C_VEL
LIN {X 0,Y 576.14,Z 662.967,A -85,B 0,C 180,E1 27183.283,E2 27183.283} C_VEL
LIN {X 0,Y 576.146,Z 662.967,A -85,B 0,C 180,E1 27180,E2 27180} C_VEL
LIN {X 0,Y 576.142,Z 662.969,A -85,B 0,C 180,E1 27176.816,E2 27176.816} C_VEL
LIN {X 0,Y 576.16,Z 662.969,A -85,B 0,C 180,E1 27173.523,E2 27173.523} C_VEL
LIN {X 0,Y 576.158,Z 662.969,A -85,B 0,C 180,E1 27170.208,E2 27170.208} C_VEL
LIN {X 0,Y 576.14,Z 662.969,A -85,B 0,C 180,E1 27166.961,E2 27166.961} C_VEL
LIN {X 0,Y 576.147,Z 662.967,A -85,B 0,C 180,E1 27163.775,E2 27163.775} C_VEL
LIN {X 0,Y 576.159,Z 662.965,A -85,B 0,C 180,E1 27163.291,E2 27163.291} C_VEL
LIN {X 0,Y 575.18,Z 663.091,A -85,B 0,C 180,E1 27162.525,E2 27162.525} C_VEL
LIN {X 0,Y 568.746,Z 663.887,A -85,B 0,C 180,E1 27160.375,E2 27160.375} C_VEL
LIN {X 0,Y 568.211,Z 663.955,A -85,B 0,C 180,E1 27159.815,E2 27159.815} C_VEL
LIN {X 0,Y 568.222,Z 663.955,A -85,B 0,C 180,E1 27156.567,E2 27156.567} C_VEL
LIN {X 0,Y 568.214,Z 663.954,A -85,B 0,C 180,E1 27153.226,E2 27153.226} C_VEL
LIN {X 0,Y 568.203,Z 663.954,A -85,B 0,C 180,E1 27149.969,E2 27149.969} C_VEL
LIN {X 0,Y 568.202,Z 663.955,A -85,B 0,C 180,E1 27146.7,E2 27146.7} C_VEL
LIN {X 0,Y 568.202,Z 663.953,A -85,B 0,C 180,E1 27143.503,E2 27143.503} C_VEL
LIN {X 0,Y 568.202,Z 663.953,A -85,B 0,C 180,E1 27140.262,E2 27140.262} C_VEL
LIN {X 0,Y 568.204,Z 663.956,A -85,B 0,C 180,E1 27137.056,E2 27137.056} C_VEL
LIN {X 0,Y 568.203,Z 663.959,A -85,B 0,C 180,E1 27133.824,E2 27133.824} C_VEL
LIN {X 0,Y 568.218,Z 663.962,A -85,B 0,C 180,E1 27130.489,E2 27130.489} C_VEL
LIN {X 0,Y 568.222,Z 663.957,A -85,B 0,C 180,E1 27127.124,E2 27127.124} C_VEL
LIN {X 0,Y 568.225,Z 663.962,A -85,B 0,C 180,E1 27126.676,E2 27126.676} C_VEL
LIN {X 0,Y 570.612,Z 670.362,A -85,B 0,C 180,E1 27126.068,E2 27126.068} C_VEL
LIN {X 0,Y 573.137,Z 676.968,A -85,B 0,C 180,E1 27125.442,E2 27125.442} C_VEL
LIN {X 0,Y 572.307,Z 723.466,A -85,B 0,C 180,E1 27122.316,E2 27122.316} C_VEL
LIN {X 0,Y 571.713,Z 766.078,A -85,B 0,C 180,E1 27119.557,E2 27119.557} C_VEL
LIN {X 0,Y 572.671,Z 773.405,A -85,B 0,C 180,E1 27119.399,E2 27119.399} C_VEL
LIN {X 0,Y 571.709,Z 1009.477,A -85,B 0,C 180,E1 27116.167,E2 27116.167} C_VEL
LIN {X 0,Y 571.536,Z 1033.914,A -85,B 0,C 180,E1 27115.771,E2 27115.771} C_VEL
LIN {X 0,Y 571.257,Z 1054.674,A -85,B 0,C 180,E1 27115.239,E2 27115.239} C_VEL
LIN {X 0,Y 570.928,Z 1074.946,A -85,B 0,C 180,E1 27114.522,E2 27114.522} C_VEL
LIN {X 0,Y 570.551,Z 1093.879,A -85,B 0,C 180,E1 27113.659,E2 27113.659} C_VEL
LIN {X 0,Y 570.127,Z 1112.944,A -85,B 0,C 180,E1 27112.585,E2 27112.585} C_VEL
LIN {X 0,Y 569.709,Z 1130.707,A -85,B 0,C 180,E1 27111.377,E2 27111.377} C_VEL
LIN {X 0,Y 569.307,Z 1148.034,A -85,B 0,C 180,E1 27109.974,E2 27109.974} C_VEL
LIN {X 0,Y 568.945,Z 1164.038,A -85,B 0,C 180,E1 27108.441,E2 27108.441} C_VEL
LIN {X 0,Y 568.633,Z 1178.905,A -85,B 0,C 180,E1 27106.76,E2 27106.76} C_VEL
LIN {X 0,Y 568.379,Z 1192.187,A -85,B 0,C 180,E1 27104.986,E2 27104.986} C_VEL
LIN {X 0,Y 568.211,Z 1203.366,A -85,B 0,C 180,E1 27103.223,E2 27103.223} C_VEL
LIN {X 0,Y 568.074,Z 1213.694,A -85,B 0,C 180,E1 27101.266,E2 27101.266} C_VEL
LIN {X 0,Y 567.982,Z 1222.012,A -85,B 0,C 180,E1 27099.32,E2 27099.32} C_VEL
LIN {X 0,Y 567.929,Z 1228.876,A -85,B 0,C 180,E1 27097.282,E2 27097.282} C_VEL
LIN {X 0,Y 567.911,Z 1234.168,A -85,B 0,C 180,E1 27095.151,E2 27095.151} C_VEL
LIN {X 0,Y 567.913,Z 1237.506,A -85,B 0,C 180,E1 27093.128,E2 27093.128} C_VEL
LIN {X 0,Y 567.913,Z 1239.241,A -85,B 0,C 180,E1 27091.109,E2 27091.109} C_VEL
LIN {X 0,Y 567.914,Z 1239.294,A -85,B 0,C 180,E1 27088.991,E2 27088.991} C_VEL
LIN {X 0,Y 567.914,Z 1237.718,A -85,B 0,C 180,E1 27086.972,E2 27086.972} C_VEL
LIN {X 0,Y 567.912,Z 1234.348,A -85,B 0,C 180,E1 27084.848,E2 27084.848} C_VEL
LIN {X 0,Y 567.927,Z 1229.441,A -85,B 0,C 180,E1 27082.819,E2 27082.819} C_VEL
LIN {X 0,Y 567.972,Z 1222.762,A -85,B 0,C 180,E1 27080.781,E2 27080.781} C_VEL
LIN {X 0,Y 568.063,Z 1214.578,A -85,B 0,C 180,E1 27078.836,E2 27078.836} C_VEL
LIN {X 0,Y 568.172,Z 1205.017,A -85,B 0,C 180,E1 27076.982,E2 27076.982} C_VEL
LIN {X 0,Y 568.356,Z 1193.495,A -85,B 0,C 180,E1 27075.117,E2 27075.117} C_VEL
LIN {X 0,Y 568.598,Z 1180.473,A -85,B 0,C 180,E1 27073.343,E2 27073.343} C_VEL
LIN {X 0,Y 568.907,Z 1165.605,A -85,B 0,C 180,E1 27071.633,E2 27071.633} C_VEL
LIN {X 0,Y 569.264,Z 1149.634,A -85,B 0,C 180,E1 27070.078,E2 27070.078} C_VEL
LIN {X 0,Y 569.665,Z 1132.905,A -85,B 0,C 180,E1 27068.695,E2 27068.695} C_VEL
LIN {X 0,Y 570.091,Z 1115.526,A -85,B 0,C 180,E1 27067.483,E2 27067.483} C_VEL
LIN {X 0,Y 570.492,Z 1096.63,A -85,B 0,C 180,E1 27066.392,E2 27066.392} C_VEL
LIN {X 0,Y 570.87,Z 1077.004,A -85,B 0,C 180,E1 27065.474,E2 27065.474} C_VEL
LIN {X 0,Y 571.227,Z 1056.493,A -85,B 0,C 180,E1 27064.728,E2 27064.728} C_VEL
LIN {X 0,Y 571.525,Z 1035.455,A -85,B 0,C 180,E1 27064.172,E2 27064.172} C_VEL
LIN {X 0,Y 571.698,Z 1012.312,A -85,B 0,C 180,E1 27063.781,E2 27063.781} C_VEL
LIN {X 0,Y 572.667,Z 775.812,A -85,B 0,C 180,E1 27060.545,E2 27060.545} C_VEL
LIN {X 0,Y 570.871,Z 767.455,A -85,B 0,C 180,E1 27060.311,E2 27060.311} C_VEL
LIN {X 0,Y 571.505,Z 733.67,A -85,B 0,C 180,E1 27057.156,E2 27057.156} C_VEL
LIN {X 0,Y 572.156,Z 700.936,A -85,B 0,C 180,E1 27054.009,E2 27054.009} C_VEL
LIN {X 0,Y 572.361,Z 675.888,A -85,B 0,C 180,E1 27051.581,E2 27051.581} C_VEL
LIN {X 0,Y 568.221,Z 663.96,A -85,B 0,C 180,E1 27050.103,E2 27050.103} C_VEL
LIN {X 0,Y 568.213,Z 663.955,A -85,B 0,C 180,E1 27046.664,E2 27046.664} C_VEL
LIN {X 0,Y 568.205,Z 663.953,A -85,B 0,C 180,E1 27043.336,E2 27043.336} C_VEL
LIN {X 0,Y 568.219,Z 663.954,A -85,B 0,C 180,E1 27040.053,E2 27040.053} C_VEL
LIN {X 0,Y 568.202,Z 663.955,A -85,B 0,C 180,E1 27036.748,E2 27036.748} C_VEL
LIN {X 0,Y 568.215,Z 664.048,A -85,B 0,C 180,E1 27033.556,E2 27033.556} C_VEL
LIN {X 0,Y 572.235,Z 675.539,A -85,B 0,C 180,E1 27032.254,E2 27032.254} C_VEL
LIN {X 0,Y 571.274,Z 713.39,A -85,B 0,C 180,E1 27029.058,E2 27029.058} C_VEL
LIN {X 0,Y 570.592,Z 753.778,A -85,B 0,C 180,E1 27025.814,E2 27025.814} C_VEL
LIN {X 0,Y 570.009,Z 794.213,A -85,B 0,C 180,E1 27022.646,E2 27022.646} C_VEL
LIN {X 0,Y 569.479,Z 836.79,A -85,B 0,C 180,E1 27019.38,E2 27019.38} C_VEL
LIN {X 0,Y 569.465,Z 845.324,A -85,B 0,C 180,E1 27018.762,E2 27018.762} C_VEL
LIN {X 0,Y 570.055,Z 852.006,A -85,B 0,C 180,E1 27018.653,E2 27018.653} C_VEL
LIN {X 0,Y 569.596,Z 1014.903,A -85,B 0,C 180,E1 27016.518,E2 27016.518} C_VEL
LIN {X 0,Y 569.46,Z 1032.883,A -85,B 0,C 180,E1 27016.09,E2 27016.09} C_VEL
LIN {X 0,Y 569.273,Z 1048.9,A -85,B 0,C 180,E1 27015.522,E2 27015.522} C_VEL
LIN {X 0,Y 569.065,Z 1064.098,A -85,B 0,C 180,E1 27014.812,E2 27014.812} C_VEL
LIN {X 0,Y 568.834,Z 1079.752,A -85,B 0,C 180,E1 27013.883,E2 27013.883} C_VEL
LIN {X 0,Y 568.608,Z 1094.164,A -85,B 0,C 180,E1 27012.801,E2 27012.801} C_VEL
LIN {X 0,Y 568.411,Z 1107.115,A -85,B 0,C 180,E1 27011.62,E2 27011.62} C_VEL
LIN {X 0,Y 568.232,Z 1119.489,A -85,B 0,C 180,E1 27010.237,E2 27010.237} C_VEL
LIN {X 0,Y 568.102,Z 1129.864,A -85,B 0,C 180,E1 27008.808,E2 27008.808} C_VEL
LIN {X 0,Y 568.014,Z 1138.886,A -85,B 0,C 180,E1 27007.281,E2 27007.281} C_VEL
LIN {X 0,Y 567.951,Z 1146.78,A -85,B 0,C 180,E1 27005.557,E2 27005.557} C_VEL
LIN {X 0,Y 567.929,Z 1152.33,A -85,B 0,C 180,E1 27003.937,E2 27003.937} C_VEL
LIN {X 0,Y 567.915,Z 1156.463,A -85,B 0,C 180,E1 27002.22,E2 27002.22} C_VEL
LIN {X 0,Y 567.916,Z 1158.792,A -85,B 0,C 180,E1 27000.505,E2 27000.505} C_VEL
LIN {X 0,Y 567.913,Z 1159.464,A -85,B 0,C 180,E1 26998.79,E2 26998.79} C_VEL
LIN {X 0,Y 567.914,Z 1158.365,A -85,B 0,C 180,E1 26996.973,E2 26996.973} C_VEL
LIN {X 0,Y 567.921,Z 1155.437,A -85,B 0,C 180,E1 26995.191,E2 26995.191} C_VEL
LIN {X 0,Y 567.931,Z 1151,A -85,B 0,C 180,E1 26993.531,E2 26993.531} C_VEL
LIN {X 0,Y 567.967,Z 1144.502,A -85,B 0,C 180,E1 26991.802,E2 26991.802} C_VEL
LIN {X 0,Y 568.024,Z 1136.908,A -85,B 0,C 180,E1 26990.272,E2 26990.272} C_VEL
LIN {X 0,Y 568.122,Z 1128.108,A -85,B 0,C 180,E1 26988.838,E2 26988.838} C_VEL
LIN {X 0,Y 568.277,Z 1116.366,A -85,B 0,C 180,E1 26987.295,E2 26987.295} C_VEL
LIN {X 0,Y 568.45,Z 1104.184,A -85,B 0,C 180,E1 26986.004,E2 26986.004} C_VEL
LIN {X 0,Y 568.669,Z 1090.533,A -85,B 0,C 180,E1 26984.813,E2 26984.813} C_VEL
LIN {X 0,Y 568.899,Z 1075.801,A -85,B 0,C 180,E1 26983.773,E2 26983.773} C_VEL
LIN {X 0,Y 569.112,Z 1060.995,A -85,B 0,C 180,E1 26982.939,E2 26982.939} C_VEL
LIN {X 0,Y 569.344,Z 1044.456,A -85,B 0,C 180,E1 26982.208,E2 26982.208} C_VEL
LIN {X 0,Y 569.511,Z 1027.178,A -85,B 0,C 180,E1 26981.665,E2 26981.665} C_VEL
LIN {X 0,Y 569.635,Z 1010.618,A -85,B 0,C 180,E1 26981.32,E2 26981.32} C_VEL
LIN {X 0,Y 569.856,Z 847.975,A -85,B 0,C 180,E1 26979.197,E2 26979.197} C_VEL
LIN {X 0,Y 569.407,Z 844.534,A -85,B 0,C 180,E1 26979.117,E2 26979.117} C_VEL
LIN {X 0,Y 569.945,Z 799.946,A -85,B 0,C 180,E1 26975.708,E2 26975.708} C_VEL
LIN {X 0,Y 570.558,Z 756.72,A -85,B 0,C 180,E1 26972.329,E2 26972.329} C_VEL
LIN {X 0,Y 571.25,Z 717.159,A -85,B 0,C 180,E1 26969.147,E2 26969.147} C_VEL
LIN {X 0,Y 574.673,Z 693.823,A -85,B 0,C 180,E1 26966.707,E2 26966.707} C_VEL
LIN {X 0,Y 577.765,Z 680.378,A -85,B 0,C 180,E1 26965.189,E2 26965.189} C_VEL
LIN {X 0,Y 575.737,Z 677.428,A -85,B 0,C 180,E1 26963.687,E2 26963.687} C_VEL
LIN {X 0,Y 575.456,Z 676.061,A -85,B 0,C 180,E1 26962.546,E2 26962.546} C_VEL
LIN {X 0,Y 575.605,Z 676.719,A -85,B 0,C 180,E1 26961.735,E2 26961.735} C_VEL
LIN {X 0,Y 576.224,Z 678.613,A -85,B 0,C 180,E1 26961.056,E2 26961.056} C_VEL
LIN {X 0,Y 573.551,Z 689.827,A -85,B 0,C 180,E1 26960.225,E2 26960.225} C_VEL
LIN {X 0,Y 571.809,Z 705.489,A -85,B 0,C 180,E1 26959.257,E2 26959.257} C_VEL
LIN {X 0,Y 570.77,Z 733.022,A -85,B 0,C 180,E1 26957.771,E2 26957.771} C_VEL
LIN {X 0,Y 571.613,Z 754.211,A -85,B 0,C 180,E1 26956.649,E2 26956.649} C_VEL
LIN {X 0,Y 573.717,Z 767.803,A -85,B 0,C 180,E1 26955.892,E2 26955.892} C_VEL
LIN {X 0,Y 577.121,Z 778.728,A -85,B 0,C 180,E1 26955.231,E2 26955.231} C_VEL
LIN {X 0,Y 581.366,Z 786.887,A -85,B 0,C 180,E1 26954.671,E2 26954.671} C_VEL
LIN {X 0,Y 585.737,Z 792.393,A -85,B 0,C 180,E1 26954.198,E2 26954.198} C_VEL
LIN {X 0,Y 589.345,Z 795.568,A -85,B 0,C 180,E1 26953.72,E2 26953.72} C_VEL
LIN {X 0,Y 592.373,Z 797.278,A -85,B 0,C 180,E1 26953.184,E2 26953.184} C_VEL
LIN {X 0,Y 594.683,Z 797.543,A -85,B 0,C 180,E1 26952.573,E2 26952.573} C_VEL
LIN {X 0,Y 595.786,Z 796.371,A -85,B 0,C 180,E1 26951.974,E2 26951.974} C_VEL
LIN {X 0,Y 595.645,Z 793.952,A -85,B 0,C 180,E1 26951.405,E2 26951.405} C_VEL
LIN {X 0,Y 594.301,Z 790.455,A -85,B 0,C 180,E1 26950.908,E2 26950.908} C_VEL
LIN {X 0,Y 591.7,Z 785.738,A -85,B 0,C 180,E1 26950.49,E2 26950.49} C_VEL
LIN {X 0,Y 587.782,Z 777.673,A -85,B 0,C 180,E1 26950.04,E2 26950.04} C_VEL
LIN {X 0,Y 584.818,Z 768.119,A -85,B 0,C 180,E1 26949.694,E2 26949.694} C_VEL
LIN {X 0,Y 582.847,Z 756.946,A -85,B 0,C 180,E1 26949.46,E2 26949.46} C_VEL
LIN {X 0,Y 581.87,Z 743.293,A -85,B 0,C 180,E1 26949.343,E2 26949.343} C_VEL
LIN {X 0,Y 581.756,Z 687.692,A -85,B 0,C 180,E1 26949.329,E2 26949.329} C_VEL
LIN {X 0,Y 578.208,Z 693.754,A -85,B 0,C 180,E1 26948.898,E2 26948.898} C_VEL
LIN {X 0,Y 575.939,Z 695.845,A -85,B 0,C 180,E1 26948.617,E2 26948.617} C_VEL
LIN {X 0,Y 574.37,Z 696.004,A -85,B 0,C 180,E1 26948.407,E2 26948.407} C_VEL
LIN {X 0,Y 573.366,Z 749.957,A -85,B 0,C 180,E1 26945.129,E2 26945.129} C_VEL
LIN {X 0,Y 573.331,Z 759.539,A -85,B 0,C 180,E1 26944.583,E2 26944.583} C_VEL
LIN {X 0,Y 574.381,Z 767.418,A -85,B 0,C 180,E1 26944.394,E2 26944.394} C_VEL
LIN {X 0,Y 573.219,Z 1001.468,A -85,B 0,C 180,E1 26941.057,E2 26941.057} C_VEL
LIN {X 0,Y 572.864,Z 1066.103,A -85,B 0,C 180,E1 26940.123,E2 26940.123} C_VEL
LIN {X 0,Y 572.551,Z 1088.393,A -85,B 0,C 180,E1 26939.603,E2 26939.603} C_VEL
LIN {X 0,Y 572.129,Z 1110.433,A -85,B 0,C 180,E1 26938.89,E2 26938.89} C_VEL
LIN {X 0,Y 571.7,Z 1131.685,A -85,B 0,C 180,E1 26938.002,E2 26938.002} C_VEL
LIN {X 0,Y 571.187,Z 1151.75,A -85,B 0,C 180,E1 26936.961,E2 26936.961} C_VEL
LIN {X 0,Y 570.675,Z 1171.156,A -85,B 0,C 180,E1 26935.755,E2 26935.755} C_VEL
LIN {X 0,Y 570.181,Z 1189.795,A -85,B 0,C 180,E1 26934.392,E2 26934.392} C_VEL
LIN {X 0,Y 569.67,Z 1208.073,A -85,B 0,C 180,E1 26932.824,E2 26932.824} C_VEL
LIN {X 0,Y 569.242,Z 1224.189,A -85,B 0,C 180,E1 26931.213,E2 26931.213} C_VEL
LIN {X 0,Y 568.857,Z 1239.882,A -85,B 0,C 180,E1 26929.403,E2 26929.403} C_VEL
LIN {X 0,Y 568.558,Z 1254.046,A -85,B 0,C 180,E1 26927.501,E2 26927.501} C_VEL
LIN {X 0,Y 568.318,Z 1266.743,A -85,B 0,C 180,E1 26925.511,E2 26925.511} C_VEL
LIN {X 0,Y 568.141,Z 1277.856,A -85,B 0,C 180,E1 26923.433,E2 26923.433} C_VEL
LIN {X 0,Y 568.027,Z 1287.488,A -85,B 0,C 180,E1 26921.268,E2 26921.268} C_VEL
LIN {X 0,Y 567.967,Z 1295.231,A -85,B 0,C 180,E1 26919.117,E2 26919.117} C_VEL
LIN {X 0,Y 567.924,Z 1300.904,A -85,B 0,C 180,E1 26917.079,E2 26917.079} C_VEL
LIN {X 0,Y 567.907,Z 1305.556,A -85,B 0,C 180,E1 26914.798,E2 26914.798} C_VEL
LIN {X 0,Y 567.899,Z 1308.318,A -85,B 0,C 180,E1 26912.624,E2 26912.624} C_VEL
LIN {X 0,Y 567.894,Z 1309.395,A -85,B 0,C 180,E1 26910.505,E2 26910.505} C_VEL
LIN {X 0,Y 567.898,Z 1308.892,A -85,B 0,C 180,E1 26908.184,E2 26908.184} C_VEL
LIN {X 0,Y 567.898,Z 1306.858,A -85,B 0,C 180,E1 26906.063,E2 26906.063} C_VEL
LIN {X 0,Y 567.906,Z 1303.199,A -85,B 0,C 180,E1 26903.937,E2 26903.937} C_VEL
LIN {X 0,Y 567.936,Z 1297.533,A -85,B 0,C 180,E1 26901.651,E2 26901.651} C_VEL
LIN {X 0,Y 567.988,Z 1291.048,A -85,B 0,C 180,E1 26899.657,E2 26899.657} C_VEL
LIN {X 0,Y 568.074,Z 1282.693,A -85,B 0,C 180,E1 26897.601,E2 26897.601} C_VEL
LIN {X 0,Y 568.22,Z 1272.542,A -85,B 0,C 180,E1 26895.531,E2 26895.531} C_VEL
LIN {X 0,Y 568.41,Z 1261.623,A -85,B 0,C 180,E1 26893.654,E2 26893.654} C_VEL
LIN {X 0,Y 568.679,Z 1248.033,A -85,B 0,C 180,E1 26891.657,E2 26891.657} C_VEL
LIN {X 0,Y 569.02,Z 1232.809,A -85,B 0,C 180,E1 26889.748,E2 26889.748} C_VEL
LIN {X 0,Y 569.43,Z 1217.028,A -85,B 0,C 180,E1 26888.038,E2 26888.038} C_VEL
LIN {X 0,Y 569.927,Z 1199.022,A -85,B 0,C 180,E1 26886.368,E2 26886.368} C_VEL
LIN {X 0,Y 570.428,Z 1180.491,A -85,B 0,C 180,E1 26884.902,E2 26884.902} C_VEL
LIN {X 0,Y 570.94,Z 1161.009,A -85,B 0,C 180,E1 26883.589,E2 26883.589} C_VEL
LIN {X 0,Y 571.46,Z 1140.541,A -85,B 0,C 180,E1 26882.434,E2 26882.434} C_VEL
LIN {X 0,Y 571.962,Z 1120.272,A -85,B 0,C 180,E1 26881.496,E2 26881.496} C_VEL
LIN {X 0,Y 572.349,Z 1098.64,A -85,B 0,C 180,E1 26880.704,E2 26880.704} C_VEL
LIN {X 0,Y 572.74,Z 1076.503,A -85,B 0,C 180,E1 26880.095,E2 26880.095} C_VEL
LIN {X 0,Y 572.962,Z 1054.213,A -85,B 0,C 180,E1 26879.682,E2 26879.682} C_VEL
